# B&R Automation Studio project NewPendant_NG4_11_05_25A (part 4)

```c
	node[i].pHeadNode	= (UDINT)&node[P_MODE_TVL_CALIB];
	node[i].Type = N_EDIT;
	node[i].var.Type = T_SCALED;
	node[i].var.Var1ID = parGEN_CalibTime4;
	//strcpy(node[i++].var.Format, "(4)Time High Vel. REV:   %s");
	strcpy(node[i++].var.Format, "%name%: %s");

	node[i].pHeadNode	= (UDINT)&node[P_MODE_TVL_CALIB];
	node[i].Type = N_SCROLL +  N_EVENT ;
	node[i].Event = EVNT_OK;
	node[i].var.Type = T_STRING;
	node[i].var.Var1ID = (h++);
	strcpy(node[i++].var.Format, " %s");

	// P_MODE_TVL_CALIB_VER
	i= P_MODE_TVL_CALIB_VER;			h=varSTRING_HMI_0;
	SetPageDict(&cfg->PagesDict[n++] , P_MODE_TVL_CALIB_VER , "P_MODE_TVL_CALIB_VER");

	node[i].pHeadNode	= (UDINT)&node[P_MODE_TVL_CALIB_VER];
	node[i].Type = N_SCROLL +  N_EVENT ;
	node[i].Event = EVNT_CANCEL;
	strcpy(node[i++].var.Format, "Repeat !!!");	//ActPos:

	node[i].pHeadNode	= (UDINT)&node[P_MODE_TVL_CALIB_VER];
	node[i].Type = N_SCROLL;
	node[i].var.Type = T_STRING;
	node[i].var.Var1ID = (h++);
	strcpy(node[i++].var.Format, "%s");

	node[i].pHeadNode	= (UDINT)&node[P_MODE_TVL_CALIB_VER];
	node[i].Type = N_SCROLL;
	node[i].var.Type = T_STRING;
	node[i].var.Var1ID = (h++);
	strcpy(node[i++].var.Format, "%s");

	node[i].pHeadNode	= (UDINT)&node[P_MODE_TVL_CALIB_VER];
	node[i].Type = N_SCROLL;
	node[i].var.Type = T_STRING;
	node[i].var.Var1ID = (h++);
	strcpy(node[i++].var.Format, "%s");

	node[i].pHeadNode	= (UDINT)&node[P_MODE_TVL_CALIB_VER];
	node[i].Type = N_SCROLL +  N_EVENT ;
	node[i].Event = EVNT_OK;
	//node[i].var.Type = T_STRING;
	//node[i].var.Var1ID = (h++);
	//strcpy(node[i++].var.Format, "%s");
	strcpy(node[i++].var.Format, "Save Calibration !!!");

	///////////////////////////////////////

	i= P_MODE_TRACK_CALIB_PAR;			h=varSTRING_HMI_0;
	SetPageDict(&cfg->PagesDict[n++] , P_MODE_TRACK_CALIB_PAR , "P_MODE_TRACK_CALIB_PAR");

	node[i].pHeadNode	= (UDINT)&node[P_MODE_TRACK_CALIB_PAR];
	node[i].Type = N_SCROLL + N_EVENT;
	node[i].Event = EVNT_CANCEL;
	node[i].var.Type = T_STRING;
	node[i].var.Var1ID = (h++);
	strcpy(node[i++].var.Format, "%s");

	node[i].pHeadNode	= (UDINT)&node[P_MODE_TRACK_CALIB_PAR];
	node[i].Type = N_SCROLL + N_EDIT_IN_PLACE;
	node[i].var.Type = T_STRING;
	node[i].var.Var1ID = (h++);
	strcpy(node[i++].var.Format, "%s");

	node[i].pHeadNode	= (UDINT)&node[P_MODE_TRACK_CALIB_PAR];
	node[i].Type = N_EDIT;
	node[i].var.Type = T_SCALED;
	node[i].var.Var1ID = parGEN_Radius;
	strcpy(node[i++].var.Format, "%name%: %s");

	node[i].pHeadNode	= (UDINT)&node[P_MODE_TRACK_CALIB_PAR];
	node[i].Type = N_EDIT;
	node[i].var.Type = T_SCALED;
	node[i].var.Var1ID = parTVL_POS_OFFSET;
	strcpy(node[i++].var.Format, "%name%: %s");

	node[i].pHeadNode	= (UDINT)&node[P_MODE_TRACK_CALIB_PAR];
	node[i].Type = N_SCROLL + N_EVENT;
	node[i].Event = EVNT_OK;
	node[i].var.Type = T_STRING;
	node[i].var.Var1ID = (h++);
	strcpy(node[i++].var.Format, "%s");

	node[i].pHeadNode	= (UDINT)&node[P_MODE_TRACK_CALIB_PAR];
	node[i].Type = N_SCROLL + N_EVENT;
	node[i].Event = EVNT_ACKN;
	node[i].var.Type = T_STRING;
	node[i].var.Var1ID = (h++);
	strcpy(node[i++].var.Format, "%s");

	// P_MODE_TRACK_CALIB_PAR
	i= P_MODE_TRACK_CALIB;			h=varSTRING_HMI_0;
	SetPageDict(&cfg->PagesDict[n++] , P_MODE_TRACK_CALIB, "P_MODE_TRACK_CALIB");

	node[i].pHeadNode	= (UDINT)&node[P_MODE_TRACK_CALIB];
	node[i].Type = N_SCROLL + N_EVENT;
	node[i].Event = EVNT_CANCEL;
	node[i].var.Type = T_STRING;
	node[i].var.Var1ID = (h++);
	strcpy(node[i++].var.Format, "%s");

	node[i].pHeadNode	= (UDINT)&node[P_MODE_TRACK_CALIB];
	node[i].Type = N_SCROLL + N_EVENT;
	node[i].Event = EVNT_ACKN;
	node[i].var.Type = T_STRING;
	node[i].var.Var1ID = (h++);
	strcpy(node[i++].var.Format, "%s");

	node[i].pHeadNode	= (UDINT)&node[P_MODE_TRACK_CALIB];
	node[i].Type = N_SCROLL;
	node[i].var.Type = T_STRING;
	node[i].var.Var1ID = (h++);
	strcpy(node[i++].var.Format, "%s");

	node[i].pHeadNode	= (UDINT)&node[P_MODE_TRACK_CALIB];
	node[i].Type = N_SCROLL;
	node[i].var.Type = T_STRING;
	node[i].var.Var1ID = (h++);
	strcpy(node[i++].var.Format, "%s");

	node[i].pHeadNode	= (UDINT)&node[P_MODE_TRACK_CALIB];
	node[i].Type = N_SCROLL;
	node[i].var.Type = T_STRING;
	node[i].var.Var1ID = (h++);
	strcpy(node[i++].var.Format, "%s");

	node[i].pHeadNode	= (UDINT)&node[P_MODE_TRACK_CALIB];
	node[i].Type = N_SCROLL + N_EVENT;
	node[i].Event = EVNT_ACKN_ALL;
	node[i].var.Type = T_STRING;
	node[i].var.Var1ID = (h++);
	strcpy(node[i++].var.Format, "%s");

	node[i].pHeadNode	= (UDINT)&node[P_MODE_TRACK_CALIB];
	node[i].Type = N_SCROLL + N_EVENT;
	node[i].Event = EVNT_OK;
	node[i].var.Type = T_STRING;
	node[i].var.Var1ID = (h++);
	strcpy(node[i++].var.Format, "%s");

	// P_MODE_TRACK_CALIB_VER
	i= P_MODE_TRACK_CALIB_VER;			h=varSTRING_HMI_0;
	SetPageDict(&cfg->PagesDict[n++] , P_MODE_TRACK_CALIB_VER , "P_MODE_TRACK_CALIB_VER");

	node[i].pHeadNode	= (UDINT)&node[P_MODE_TRACK_CALIB_VER];
	node[i].Type = N_SCROLL + N_EVENT;
	node[i].Event = EVNT_CANCEL;
	node[i].var.Type = T_STRING;
	node[i].var.Var1ID = (h++);
	strcpy(node[i++].var.Format, "%s");

	node[i].pHeadNode	= (UDINT)&node[P_MODE_TRACK_CALIB_VER];
	node[i].Type = N_SCROLL + N_EVENT;
	node[i].Event = EVNT_ACKN;
	node[i].var.Type = T_STRING;
	node[i].var.Var1ID = (h++);
	strcpy(node[i++].var.Format, "%s");

	node[i].pHeadNode	= (UDINT)&node[P_MODE_TRACK_CALIB_VER];
	node[i].Type = N_SCROLL;
	node[i].var.Type = T_STRING;
	node[i].var.Var1ID = (h++);
	strcpy(node[i++].var.Format, "%s");

	node[i].pHeadNode	= (UDINT)&node[P_MODE_TRACK_CALIB_VER];
	node[i].Type = N_SCROLL;
	node[i].var.Type = T_STRING;
	node[i].var.Var1ID = (h++);
	strcpy(node[i++].var.Format, "%s");

	node[i].pHeadNode	= (UDINT)&node[P_MODE_TRACK_CALIB_VER];
	node[i].Type = N_SCROLL;
	node[i].var.Type = T_STRING;
	node[i].var.Var1ID = (h++);
	strcpy(node[i++].var.Format, "%s");

	node[i].pHeadNode	= (UDINT)&node[P_MODE_TRACK_CALIB_VER];
	node[i].Type = N_SCROLL + N_EVENT;
	node[i].Event = EVNT_OK;
	node[i].var.Type = T_STRING;
	node[i].var.Var1ID = (h++);
	strcpy(node[i++].var.Format, "%s");

	/////////////////////////////////////

	// P_SPEC_OPERATION
	i = P_SPEC_OPERATION;			h=varSTRING_HMI_0;
	SetPageDict(&cfg->PagesDict[n++] , P_SPEC_OPERATION , "P_SPEC_OPERATION");

	node[i].pHeadNode	= (UDINT)&node[P_SPEC_OPERATION];
	node[i].Type = N_JUMP;
	node[i].JumpLineID = 0;
	node[i].pJumpNode = (UDINT)&node[P_MENU];
	strcpy(node[i++].var.Format, " Return !!!");

	node[i].pHeadNode	= (UDINT)&node[P_SPEC_OPERATION];
	node[i].Type = N_SCROLL + N_EVENT;
	node[i].Event = EVNT_SET_AMERICAN_UNIT;
	strcpy(node[i++].var.Format, "Set Default Units !");

	node[i].pHeadNode	= (UDINT)&node[P_SPEC_OPERATION];
	node[i].Type = N_SCROLL + N_EVENT;
	node[i].Event = EVNT_SET_NORMAL_UNIT;
	strcpy(node[i++].var.Format, "Set SI Units !!!");

	node[i].pHeadNode	= (UDINT)&node[P_SPEC_OPERATION];
	node[i].Type = N_SCROLL + N_EVENT;
	node[i].Event = EVNT_LOAD_DEFAULT;
	strcpy(node[i++].var.Format, "Load Defaults !!!");

	node[i].pHeadNode	= (UDINT)&node[P_SPEC_OPERATION];
	node[i].Type = N_SCROLL + N_EVENT;
	node[i].Event = EVNT_LOAD_DEFAULT_CALIB;
	strcpy(node[i++].var.Format, "Load Default Calib !");

	node[i].pHeadNode	= (UDINT)&node[P_SPEC_OPERATION];
	node[i].Type = N_SCROLL + N_EVENT;
	node[i].Event = EVNT_ENT_BTN_REQ;
	strcpy(node[i++].var.Format, "Enter Btn Req!!");

	/** P_DIAGNOSTIC **/
	 i = P_DIAGNOSTIC;			h=varSTRING_HMI_0;
	SetPageDict(&cfg->PagesDict[n++] , P_DIAGNOSTIC , "P_DIAGNOSTIC");

	node[i].pHeadNode	= (UDINT)&node[P_DIAGNOSTIC];
	node[i].Type = N_SCROLL;
	node[i].var.Type = T_STRING;
	node[i].var.Var1ID = varSTRING_MasteStepTXT;
	strcpy(node[i++].var.Format, "M: %s");

	node[i].pHeadNode	= (UDINT)&node[P_DIAGNOSTIC];
	node[i].Type = N_JUMP;
	node[i].JumpLineID = 0;
	node[i].pJumpNode = (UDINT)&node[P_DIAGN_PROC];
	strcpy(node[i++].var.Format, "Diagn PROCESS");

	node[i].pHeadNode	= (UDINT)&node[P_DIAGNOSTIC];
	node[i].Type = N_JUMP;
	node[i].JumpLineID = 0;
	node[i].pJumpNode = (UDINT)&node[P_DIAGN_TML];
	strcpy(node[i++].var.Format, "Diagn TML Servo");

	node[i].pHeadNode	= (UDINT)&node[P_DIAGNOSTIC];
	node[i].Type = N_JUMP;
	node[i].JumpLineID = 0;
	node[i].pJumpNode = (UDINT)&node[P_DIAGN_DC_MTR];
	strcpy(node[i++].var.Format, "Diagn DC Mtrs");

	node[i].pHeadNode	= (UDINT)&node[P_DIAGNOSTIC];
	node[i].Type = N_JUMP;
	node[i].JumpLineID = 0;
	node[i].pJumpNode = (UDINT)&node[P_DIAGN_AXIS];
	strcpy(node[i++].var.Format, "Diagn Axises ");

	node[i].pHeadNode	= (UDINT)&node[P_DIAGNOSTIC];
	node[i].Type = N_JUMP;
	node[i].JumpLineID = 0;
	node[i].pJumpNode = (UDINT)&node[P_DIAGN_IO];
	strcpy(node[i++].var.Format, "Diagn I/O");

	node[i].pHeadNode	= (UDINT)&node[P_DIAGNOSTIC];
	node[i].Type = N_SCROLL + N_EVENT;
	node[i].Event = EVNT_RESTART ;
	node[i].var.Type = T_STRING;
	node[i].var.Var1ID = (h++);

	strcpy(node[i++].var.Format, "RESTART !!!");

	/** P_DIAGN_TML **/
	i = P_DIAGN_TML;			h=varSTRING_HMI_0;
	SetPageDict(&cfg->PagesDict[n++] , P_DIAGN_TML , "P_DIAGN_TML");

	node[i].pHeadNode	= (UDINT)&node[P_DIAGN_TML];
	node[i].Type = N_JUMP;
	node[i].JumpLineID = 0;
	node[i].pJumpNode = (UDINT)&node[P_DIAGNOSTIC];
	strcpy(node[i++].var.Format, " Return !!!");

	node[i].pHeadNode	= (UDINT)&node[P_DIAGN_TML];
	node[i].Type =    N_SCROLL + N_EDIT_IN_PLACE;
	node[i].var.Type = T_STRING;
	node[i].var.Var1ID = (h++);

	strcpy(node[i++].var.Format,"%s");

	node[i].pHeadNode	= (UDINT)&node[P_DIAGN_TML];
	node[i].Type = N_SCROLL + N_EDIT_IN_PLACE;
	node[i].var.Type = T_STRING;
	node[i].var.Var1ID = (h++);
	strcpy(node[i++].var.Format, "Stat: %s ");

	node[i].pHeadNode	= (UDINT)&node[P_DIAGN_TML];
	node[i].Type = N_SCROLL + N_EDIT_IN_PLACE;
	node[i].var.Var1ID = (h++);
	node[i].var.Type = T_STRING;
	strcpy(node[i++].var.Format, "%s");

	node[i].pHeadNode	= (UDINT)&node[P_DIAGN_TML];
	node[i].Type = N_SCROLL +	N_EVENT ;
	node[i].Event = EVNT_TOGGLE;
	node[i].var.Type = T_STRING;
	node[i].var.Var1ID = (h++);
	strcpy(node[i++].var.Format, "%s ");

	node[i].pHeadNode	= (UDINT)&node[P_DIAGN_TML];
	node[i].Type = N_SCROLL + N_EDIT_IN_PLACE;
	node[i].var.Type = T_STRING;
	node[i].var.Var1ID = (h++);
	strcpy(node[i++].var.Format, "%s");

	node[i].pHeadNode	= (UDINT)&node[P_DIAGN_TML];
	node[i].Type = N_SCROLL + N_EDIT_IN_PLACE;
	node[i].var.Type = T_STRING;
	node[i].var.Var1ID = (h++);
	strcpy(node[i++].var.Format, "%s");

	node[i].pHeadNode	= (UDINT)&node[P_DIAGN_TML];
	node[i].Type = N_SCROLL;
	node[i].var.Var1ID = (h++);
	node[i].var.Type = T_STRING;
	strcpy(node[i++].var.Format, "%s");

	node[i].pHeadNode	= (UDINT)&node[P_DIAGN_TML];
	node[i].Type = N_SCROLL;
	node[i].var.Type = T_STRING;
	node[i].var.Var1ID = (h++);
	strcpy(node[i++].var.Format, "EnInp: %s");

	node[i].pHeadNode	= (UDINT)&node[P_DIAGN_TML];
	node[i].Type = N_SCROLL;
	node[i].var.Type = T_STRING;
	node[i].var.Var1ID = (h++);
	strcpy(node[i++].var.Format, "%s "); // Inp 0 & 1

	node[i].pHeadNode	= (UDINT)&node[P_DIAGN_TML];
	node[i].Type = N_SCROLL;
	node[i].var.Type = T_STRING;
	node[i].var.Var1ID = (h++);
	strcpy(node[i++].var.Format, "%s "); //Inp 2 & 3

	node[i].pHeadNode	= (UDINT)&node[P_DIAGN_TML];
	node[i].Type = N_SCROLL;
	node[i].var.Type = T_STRING;
	node[i].var.Var1ID = (h++);
	strcpy(node[i++].var.Format, "%s "); //Out 0 & 1

	node[i].pHeadNode	= (UDINT)&node[P_DIAGN_TML];
	node[i].Type = N_SCROLL;
	node[i].var.Type = T_STRING;
	node[i].var.Var1ID = (h++);
	strcpy(node[i++].var.Format, "%s "); //Out 4

	node[i].pHeadNode	= (UDINT)&node[P_DIAGN_TML];
	node[i].Type = N_SCROLL;
	node[i].var.Type = T_STRING;
	node[i].var.Var1ID = (h++);
	strcpy(node[i++].var.Format, "xCMD: %s ");

	node[i].pHeadNode	= (UDINT)&node[P_DIAGN_TML];
	node[i].Type = N_SCROLL;
	node[i].var.Type = T_STRING;
	node[i].var.Var1ID = (h++);
	strcpy(node[i++].var.Format, "%s "); //Fbk:

	node[i].pHeadNode	= (UDINT)&node[P_DIAGN_TML];
	node[i].Type = N_SCROLL + N_EVENT;
	strcpy(node[i++].var.Format, "Jog Fwd");

	node[i].pHeadNode	= (UDINT)&node[P_DIAGN_TML];
	node[i].Type = N_SCROLL + N_EVENT;
	strcpy(node[i++].var.Format, "Jog Rev");

	node[i].pHeadNode	= (UDINT)&node[P_DIAGN_TML];
	node[i].Type = N_SCROLL + N_EVENT;
	node[i].Event = EVNT_OK;
	node[i].var.Type = T_STRING;
	node[i].var.Var1ID = (h++);
	strcpy(node[i++].var.Format, "Set ABS Home  !!!");

	node[i].pHeadNode	= (UDINT)&node[P_DIAGN_TML];
	node[i].Type = N_SCROLL + N_EVENT;
	node[i].Event = EVNT_LOAD;
	node[i].var.Type = T_STRING;
	node[i].var.Var1ID = (h++);
	strcpy(node[i++].var.Format, "LOAD Setup !!!");

	node[i].pHeadNode	= (UDINT)&node[P_DIAGN_TML];
	node[i].Type = N_SCROLL + N_EVENT;
	node[i].Event = EVNT_RESTART;
	node[i].var.Type = T_STRING;
	node[i].var.Var1ID = (h++);
	strcpy(node[i++].var.Format, "RESTART !!!");

	/** P_DIAGN_PROC **/
	i = P_DIAGN_PROC;			h=varSTRING_HMI_0;
	SetPageDict(&cfg->PagesDict[n++] , P_DIAGN_PROC , "P_DIAGN_PROC");

	node[i].pHeadNode	= (UDINT)&node[P_DIAGN_PROC];
	node[i].Type = N_JUMP;
	node[i].JumpLineID = 0;
	node[i].pJumpNode = (UDINT)&node[P_DIAGNOSTIC];
	strcpy(node[i++].var.Format, " Return !!!");

	node[i].pHeadNode	= (UDINT)&node[P_DIAGN_PROC];
	node[i].Type =    N_SCROLL + N_EDIT_IN_PLACE;
	node[i].var.Type = T_STRING;
	node[i].var.Var1ID = (h++);

	strcpy(node[i++].var.Format,"%s");

	node[i].pHeadNode	= (UDINT)&node[P_DIAGN_PROC];
	node[i].Type = N_SCROLL;
	node[i].var.Type = T_STRING;
	node[i].var.Var1ID = (h++);
	strcpy(node[i++].var.Format, "Stat: %s ");

	node[i].pHeadNode	= (UDINT)&node[P_DIAGN_PROC];
	node[i].Type = N_SCROLL;
	node[i].var.Type = T_STRING;
	node[i].var.Var1ID = (h++);
	strcpy(node[i++].var.Format, "%s ");

	node[i].pHeadNode	= (UDINT)&node[P_DIAGN_PROC];
	node[i].Type = N_SCROLL +	N_EVENT ;
	node[i].Event = EVNT_TOGGLE;
	node[i].var.Type = T_STRING;
	node[i].var.Var1ID = (h++);
	strcpy(node[i++].var.Format, "%s ");

	node[i].pHeadNode	= (UDINT)&node[P_DIAGN_PROC];
	node[i].Type = N_SCROLL + N_EVENT;
	node[i].Event = EVNT_RESTART ;
	node[i].var.Type = T_STRING;
	strcpy(node[i++].var.Format, "RESTART !!!");

	/** P_DIAGN_DC_MTR **/
	i = P_DIAGN_DC_MTR;			h=varSTRING_HMI_0;
	SetPageDict(&cfg->PagesDict[n++] , P_DIAGN_DC_MTR , "P_DIAGN_DC_MTR");

	node[i].pHeadNode	= (UDINT)&node[P_DIAGN_DC_MTR];
	node[i].Type = N_JUMP;
	node[i].JumpLineID = 0;
	node[i].pJumpNode = (UDINT)&node[P_DIAGNOSTIC];
	strcpy(node[i++].var.Format, " Return !!!");

	node[i].pHeadNode	= (UDINT)&node[P_DIAGN_DC_MTR];
	node[i].Type =    N_SCROLL + N_EDIT_IN_PLACE;
	node[i].var.Type = T_STRING;
	node[i].var.Var1ID = (h++);

	strcpy(node[i++].var.Format,"%s");

	node[i].pHeadNode	= (UDINT)&node[P_DIAGN_DC_MTR];
	node[i].Type = N_SCROLL;
	node[i].var.Type = T_STRING;
	node[i].var.Var1ID = (h++);
	strcpy(node[i++].var.Format, "%s ");

	node[i].pHeadNode	= (UDINT)&node[P_DIAGN_DC_MTR];
	node[i].Type = N_SCROLL +	N_EVENT ;
	node[i].Event = EVNT_TOGGLE;
	node[i].var.Type = T_STRING;
	node[i].var.Var1ID = (h++);
	strcpy(node[i++].var.Format, "%s ");

	node[i].pHeadNode	= (UDINT)&node[P_DIAGN_DC_MTR];
	node[i].Type = N_SCROLL;
	node[i].var.Type = T_STRING;
	node[i].var.Var1ID = (h++);
	strcpy(node[i++].var.Format, "Fbk: %s ");

	node[i].pHeadNode	= (UDINT)&node[P_DIAGN_DC_MTR];
	node[i].Type = N_SCROLL + N_EVENT;
	strcpy(node[i++].var.Format, "Jog Fwd");

	node[i].pHeadNode	= (UDINT)&node[P_DIAGN_DC_MTR];
	node[i].Type = N_SCROLL + N_EVENT;
	strcpy(node[i++].var.Format, "Jog Rev");

	/** P_DIAGN_AXIS **/
	i = P_DIAGN_AXIS;			h=varSTRING_HMI_0;
	SetPageDict(&cfg->PagesDict[n++] , P_DIAGN_AXIS , "P_DIAGN_AXIS");

	node[i].pHeadNode	= (UDINT)&node[P_DIAGN_AXIS];
	node[i].Type = N_JUMP;
	node[i].JumpLineID = 0;
	node[i].pJumpNode = (UDINT)&node[P_DIAGNOSTIC];
	strcpy(node[i++].var.Format, " Return !!!");

	node[i].pHeadNode	= (UDINT)&node[P_DIAGN_AXIS];
	node[i].Type =    N_SCROLL + N_EDIT_IN_PLACE;
	node[i].var.Type = T_STRING;
	node[i].var.Var1ID = (h++);

	strcpy(node[i++].var.Format,"%s");

	node[i].pHeadNode	= (UDINT)&node[P_DIAGN_AXIS];
	node[i].Type = N_SCROLL;
	node[i].var.Type = T_STRING;
	node[i].var.Var1ID = (h++);
	strcpy(node[i++].var.Format, "%s ");

	node[i].pHeadNode	= (UDINT)&node[P_DIAGN_AXIS];
	node[i].Type = N_SCROLL ;
	node[i].var.Type = T_STRING;
	node[i].var.Var1ID = (h++);
	strcpy(node[i++].var.Format, "%s ");

	node[i].pHeadNode	= (UDINT)&node[P_DIAGN_AXIS];
	node[i].Type = N_SCROLL ;
	node[i].var.Type = T_STRING;
	node[i].var.Var1ID = (h++);
	strcpy(node[i++].var.Format, "%s ");

	node[i].pHeadNode	= (UDINT)&node[P_DIAGN_AXIS];
	node[i].Type = N_SCROLL ;
	node[i].var.Type = T_STRING;
	node[i].var.Var1ID = (h++);
	strcpy(node[i++].var.Format, "%s ");

	/** P_DIAGN_IO **/
	i = P_DIAGN_IO;			h=varSTRING_HMI_0;
	SetPageDict(&cfg->PagesDict[n++] , P_DIAGN_IO , "P_DIAGN_IO");

	node[i].pHeadNode	= (UDINT)&node[P_DIAGN_IO];
	node[i].Type = N_JUMP;
	node[i].JumpLineID = 0;
	node[i].pJumpNode = (UDINT)&node[P_DIAGNOSTIC];
	strcpy(node[i++].var.Format, " Return !!!");

	node[i].pHeadNode	= (UDINT)&node[P_DIAGN_IO];
	node[i].Type = N_SCROLL;
	node[i].var.Var1ID = (h++);
	node[i].var.Type = T_STRING;

	strcpy(node[i++].var.Format, "%s");

	node[i].pHeadNode	= (UDINT)&node[P_DIAGN_IO];
	node[i].Type = N_SCROLL;
	node[i].var.Var1ID = (h++);
	node[i].var.Type = T_STRING;
	strcpy(node[i++].var.Format, "%s");

	node[i].pHeadNode	= (UDINT)&node[P_DIAGN_IO];
	node[i].Type = N_SCROLL;
	node[i].var.Var1ID = (h++);
	node[i].var.Type = T_STRING;
	strcpy(node[i++].var.Format, "%s");

	node[i].pHeadNode	= (UDINT)&node[P_DIAGN_IO];
	node[i].Type = N_SCROLL;
	node[i].var.Var1ID = (h++);
	node[i].var.Type = T_STRING;
	strcpy(node[i++].var.Format, "%s");

	node[i].pHeadNode	= (UDINT)&node[P_DIAGN_IO];
	node[i].Type = N_SCROLL;
	node[i].var.Var1ID = (h++);
	node[i].var.Type = T_STRING;
	strcpy(node[i++].var.Format, "%s");

	node[i].pHeadNode	= (UDINT)&node[P_DIAGN_IO];
	node[i].Type = N_SCROLL;
	node[i].var.Var1ID = (h++);
	node[i].var.Type = T_STRING;
	strcpy(node[i++].var.Format, "%s");

	node[i].pHeadNode	= (UDINT)&node[P_DIAGN_IO];
	node[i].Type = N_SCROLL;
	node[i].var.Var1ID = (h++);
	node[i].var.Type = T_STRING;
	strcpy(node[i++].var.Format, "%s");

	node[i].pHeadNode	= (UDINT)&node[P_DIAGN_IO];
	node[i].Type = N_SCROLL;
	node[i].var.Var1ID = (h++);
	node[i].var.Type = T_STRING;
	strcpy(node[i++].var.Format, "%s");

	node[i].pHeadNode	= (UDINT)&node[P_DIAGN_IO];
	node[i].Type = N_SCROLL;
	node[i].var.Var1ID = (h++);
	node[i].var.Type = T_STRING;
	strcpy(node[i++].var.Format, "%s");

	node[i].pHeadNode	= (UDINT)&node[P_DIAGN_IO];
	node[i].Type = N_SCROLL;
	node[i].var.Var1ID = (h++);
	node[i].var.Type = T_STRING;
	strcpy(node[i++].var.Format, "%s");

	node[i].pHeadNode	= (UDINT)&node[P_DIAGN_IO];
	node[i].Type = N_SCROLL;
	node[i].var.Var1ID = (h++);
	node[i].var.Type = T_STRING;
	strcpy(node[i++].var.Format, "%s");

	/** P_LOGS **/
	 i = P_LOGS;			h=varSTRING_HMI_0;
	SetPageDict(&cfg->PagesDict[n++] , P_LOGS , "P_LOGS");

	node[i].pHeadNode	= (UDINT)&node[P_LOGS];
	node[i].Type = N_SCROLL + N_EDIT_IN_PLACE;
	node[i].var.Var1ID = (h++);
	node[i].var.Type = T_STRING;
	strcpy(node[i++].var.Format, "%s");

	node[i].pHeadNode	= (UDINT)&node[P_LOGS];
	node[i].Type = N_SCROLL + N_EDIT_IN_PLACE;
	node[i].var.Var1ID = (h++);
	node[i].var.Type = T_STRING;
	strcpy(node[i++].var.Format, "%s");

	node[i].pHeadNode	= (UDINT)&node[P_LOGS];
	node[i].Type = N_SCROLL + N_EDIT_IN_PLACE;
	node[i].var.Var1ID = (h++);
	node[i].var.Type = T_STRING;
	strcpy(node[i++].var.Format, "%s");

	node[i].pHeadNode	= (UDINT)&node[P_LOGS];
	node[i].Type = N_SCROLL + N_EDIT_IN_PLACE;
	node[i].var.Var1ID = (h++);
	node[i].var.Type = T_STRING;
	strcpy(node[i++].var.Format, "%s");

	node[i].pHeadNode	= (UDINT)&node[P_LOGS];
	node[i].Type = N_SCROLL + N_EDIT_IN_PLACE;
	node[i].var.Var1ID = (h++);
	node[i].var.Type = T_STRING;
	strcpy(node[i++].var.Format, "%s");

	node[i].pHeadNode	= (UDINT)&node[P_LOGS];
	node[i].Type = N_SCROLL + N_EDIT_IN_PLACE;
	node[i].var.Var1ID = (h++);
	node[i].var.Type = T_STRING;
	strcpy(node[i++].var.Format, "%s");

	/** P_ERRORS **/
	 i = P_ERRORS;			h=varSTRING_HMI_0;
	SetPageDict(&cfg->PagesDict[n++] , P_ERRORS , "P_ERRORS");

	node[i].pHeadNode	= (UDINT)&node[P_ERRORS];
	node[i].Type = N_SCROLL + N_EDIT_IN_PLACE;
	node[i].var.Var1ID = (h++);
	node[i].var.Type = T_STRING;
	strcpy(node[i++].var.Format, "%s");

	node[i].pHeadNode	= (UDINT)&node[P_ERRORS];
	node[i].Type = N_SCROLL + N_EDIT_IN_PLACE;
	node[i].var.Var1ID = (h++);
	node[i].var.Type = T_STRING;
	strcpy(node[i++].var.Format, "%s");

	node[i].pHeadNode	= (UDINT)&node[P_ERRORS];
	node[i].Type = N_SCROLL + N_EDIT_IN_PLACE;
	node[i].var.Var1ID = (h++);
	node[i].var.Type = T_STRING;
	strcpy(node[i++].var.Format, "  %s");

	node[i].pHeadNode	= (UDINT)&node[P_ERRORS];
	node[i].Type = N_SCROLL + N_EDIT_IN_PLACE;
	node[i].var.Var1ID = (h++);
	node[i].var.Type = T_STRING;
	strcpy(node[i++].var.Format, "  %s");

	node[i].pHeadNode	= (UDINT)&node[P_ERRORS];
	node[i].Type = N_SCROLL + N_EDIT_IN_PLACE;
	node[i].var.Var1ID = (h++);
	node[i].var.Type = T_STRING;
	strcpy(node[i++].var.Format, "  %s");

	node[i].pHeadNode	= (UDINT)&node[P_ERRORS];
	node[i].Type = N_SCROLL + N_EVENT;
	node[i].Event = EVNT_ACKN_ALL;
	strcpy(node[i++].var.Format, " ACK All Errors !!!");

	//////////////////////////////////////////////////////////
	//////////    FOR TESTING ONLY -

	/** P_PAR_REVIEW **/
	i = P_PAR_REVIEW;			h=varSTRING_HMI_0;
	SetPageDict(&cfg->PagesDict[n++] , P_PAR_REVIEW , "P_PAR_REVIEW");

	node[i].pHeadNode	= (UDINT)&node[P_PAR_REVIEW];
	node[i].Type = N_JUMP;
	node[i].JumpLineID = 0;
	node[i].pJumpNode = (UDINT)&node[P_MENU];
	strcpy(node[i++].var.Format, "Return ");

	node[i].pHeadNode	= (UDINT)&node[P_PAR_REVIEW];
	node[i].Type = N_SCROLL;
	strcpy(node[i++].var.Format, "**** AVC *****");

	node[i].pHeadNode	= (UDINT)&node[P_PAR_REVIEW];
	node[i].Type = N_EDIT;
	node[i].MinUserLevel = USER_OPERATOR;
	node[i].var.Type = T_SCALED;
	node[i].var.Var1ID = parAVC_StartDly;
	//strcpy(node[i++].var.Format, "AVC UpslopeDly %s");
	strcpy(node[i++].var.Format, "%name%: %s");

	node[i].pHeadNode	= (UDINT)&node[P_PAR_REVIEW];
	node[i].Type = N_EDIT;
	node[i].MinUserLevel = USER_OPERATOR;
	node[i].var.Type = T_SCALED;
	node[i].var.Var1ID = parAVC_Upslope;
	//strcpy(node[i++].var.Format, "AVC Upslope %s");
	strcpy(node[i++].var.Format, "%name%: %s");

	node[i].pHeadNode	= (UDINT)&node[P_PAR_REVIEW];
	node[i].Type = N_EDIT;
	node[i].MinUserLevel = USER_OPERATOR;
	node[i].var.Type = T_SCALED;
	node[i].var.Var1ID = parAVC_StopDly;
	//strcpy(node[i++].var.Format, "AVC StopDly %s");
	strcpy(node[i++].var.Format, "%name%: %s");

	node[i].pHeadNode	= (UDINT)&node[P_PAR_REVIEW];
	node[i].Type = N_EDIT;
	node[i].MinUserLevel = USER_OPERATOR;
	node[i].var.Type = T_SCALED;
	node[i].var.Var1ID = parAVC_DownSlope;
	//strcpy(node[i++].var.Format, "AVC DownSlope %s");
	strcpy(node[i++].var.Format, "%name%: %s");

	node[i].pHeadNode	= (UDINT)&node[P_PAR_REVIEW];
	node[i].Type = N_EDIT;
	node[i].MinUserLevel = USER_OPERATOR;
	node[i].var.Type = T_SCALED;
	node[i].var.Var1ID = parAVC_HoldTm;
	//strcpy(node[i++].var.Format, "AVC HoldTm %s");
	strcpy(node[i++].var.Format, "%name%: %s");

	node[i].pHeadNode	= (UDINT)&node[P_PAR_REVIEW];
	node[i].Type = N_SCROLL;
	strcpy(node[i++].var.Format, "**** TVL *****");

	node[i].pHeadNode	= (UDINT)&node[P_PAR_REVIEW];
	node[i].Type = N_EDIT;
	node[i].MinUserLevel = USER_OPERATOR;
	node[i].var.Type = T_SCALED;
	node[i].var.Var1ID = parTVL_StartDly;
	//strcpy(node[i++].var.Format, "TVL_StartDly %s");
	strcpy(node[i++].var.Format, "%name%: %s");

	node[i].pHeadNode	= (UDINT)&node[P_PAR_REVIEW];
	node[i].Type = N_EDIT;
	node[i].MinUserLevel = USER_OPERATOR;
	node[i].var.Type = T_SCALED;
	node[i].var.Var1ID = parTVL_RampUp;
	//strcpy(node[i++].var.Format, "TVL RampUp %s");
	strcpy(node[i++].var.Format, "%name%: %s");

	node[i].pHeadNode	= (UDINT)&node[P_PAR_REVIEW];
	node[i].Type = N_EDIT;
	node[i].MinUserLevel = USER_OPERATOR;
	node[i].var.Type = T_SCALED;
	node[i].var.Var1ID = parTVL_StopDly;
	//strcpy(node[i++].var.Format, "TVL StopDly %s");
	strcpy(node[i++].var.Format, "%name%: %s");

	node[i].pHeadNode	= (UDINT)&node[P_PAR_REVIEW];
	node[i].Type = N_EDIT;
	node[i].MinUserLevel = USER_OPERATOR;
	node[i].var.Type = T_SCALED;
	node[i].var.Var1ID = parTVL_RampDwn;
	//strcpy(node[i++].var.Format, "TVL RampDwn %s");
	strcpy(node[i++].var.Format, "%name%: %s");

	node[i].pHeadNode	= (UDINT)&node[P_PAR_REVIEW];
	node[i].Type = N_EDIT;
	node[i].MinUserLevel = USER_OPERATOR;
	node[i].var.Type = T_SCALED;
	node[i].var.Var1ID = parTVL_RewrapDly;
	//strcpy(node[i++].var.Format, "TVL RewrapDly %s");
	strcpy(node[i++].var.Format, "%name%: %s");

	node[i].pHeadNode	= (UDINT)&node[P_PAR_REVIEW];
	node[i].Type = N_EDIT;
	node[i].MinUserLevel = USER_OPERATOR;
	node[i].var.Type = T_SCALED;
	node[i].var.Var1ID = parTVL_OverlapDist;
	//strcpy(node[i++].var.Format, "TVL Overlap %s");
	strcpy(node[i++].var.Format, "%name%: %s");

	node[i].pHeadNode	= (UDINT)&node[P_PAR_REVIEW];
	node[i].Type = N_SCROLL;
	strcpy(node[i++].var.Format, "**** TIG AMP *****");

	node[i].pHeadNode	= (UDINT)&node[P_PAR_REVIEW];
	node[i].Type = N_EDIT;
	node[i].MinUserLevel = USER_OPERATOR;
	node[i].var.Type = T_SCALED;
	node[i].var.Var1ID = parTIG_StartDly;
	//strcpy(node[i++].var.Format, "TIG StartDly %s");
	strcpy(node[i++].var.Format, "%name%: %s");

	node[i].pHeadNode	= (UDINT)&node[P_PAR_REVIEW];
	node[i].Type = N_EDIT;
	node[i].MinUserLevel = USER_OPERATOR;
	node[i].var.Type = T_SCALED;
	node[i].var.Var1ID = parTIG_RampUp;
	//strcpy(node[i++].var.Format, "TIG RampUp %s");
	strcpy(node[i++].var.Format, "%name%: %s");

	node[i].pHeadNode	= (UDINT)&node[P_PAR_REVIEW];
	node[i].Type = N_EDIT;
	node[i].MinUserLevel = USER_OPERATOR;
	node[i].var.Type = T_SCALED;
	node[i].var.Var1ID = parTIG_StopDly;
	//strcpy(node[i++].var.Format, "TIG StopDly %s");
	strcpy(node[i++].var.Format, "%name%: %s");

	node[i].pHeadNode	= (UDINT)&node[P_PAR_REVIEW];
	node[i].Type = N_EDIT;
	node[i].MinUserLevel = USER_OPERATOR;
	node[i].var.Type = T_SCALED;
	node[i].var.Var1ID = parTIG_RampDwn;
	//strcpy(node[i++].var.Format, "TIG RampDwn %s");
	strcpy(node[i++].var.Format, "%name%: %s");

	node[i].pHeadNode	= (UDINT)&node[P_PAR_REVIEW];
	node[i].Type = N_SCROLL;
	strcpy(node[i++].var.Format, "**** OSC *****");

	node[i].pHeadNode	= (UDINT)&node[P_PAR_REVIEW];
	node[i].Type = N_EDIT;
	node[i].MinUserLevel = USER_OPERATOR;
	node[i].var.Type = T_SCALED;
	node[i].var.Var1ID = parOSC_StartDly;
	//strcpy(node[i++].var.Format, "OSC StartDly %s");
	strcpy(node[i++].var.Format, "%name%: %s");

	node[i].pHeadNode	= (UDINT)&node[P_PAR_REVIEW];
	node[i].Type = N_EDIT;
	node[i].MinUserLevel = USER_OPERATOR;
	node[i].var.Type = T_SCALED;
	node[i].var.Var1ID = parOSC_RampUp;
	//strcpy(node[i++].var.Format, "OSC RampUp %s");
	strcpy(node[i++].var.Format, "%name%: %s");

	node[i].pHeadNode	= (UDINT)&node[P_PAR_REVIEW];
	node[i].Type = N_EDIT;
	node[i].MinUserLevel = USER_OPERATOR;
	node[i].var.Type = T_SCALED;
	node[i].var.Var1ID = parOSC_StopDly;
	//strcpy(node[i++].var.Format, "OSC StopDly %s");
	strcpy(node[i++].var.Format, "%name%: %s");

	node[i].pHeadNode	= (UDINT)&node[P_PAR_REVIEW];
	node[i].Type = N_EDIT;
	node[i].MinUserLevel = USER_OPERATOR;
	node[i].var.Type = T_SCALED;
	node[i].var.Var1ID = parOSC_RampDwn;
	//strcpy(node[i++].var.Format, "OSC RampDwn %s");
	strcpy(node[i++].var.Format, "%name%: %s");

	node[i].pHeadNode	= (UDINT)&node[P_PAR_REVIEW];
	node[i].Type = N_SCROLL;
	strcpy(node[i++].var.Format, "**** WF *****");

	node[i].pHeadNode	= (UDINT)&node[P_PAR_REVIEW];
	node[i].Type = N_EDIT;
	node[i].MinUserLevel = USER_OPERATOR;
	node[i].var.Type = T_SCALED;
	node[i].var.Var1ID = parWF_StartDly;
	//strcpy(node[i++].var.Format, "parWF StartDly %s");
	strcpy(node[i++].var.Format, "%name%: %s");

	node[i].pHeadNode	= (UDINT)&node[P_PAR_REVIEW];
	node[i].Type = N_EDIT;
	node[i].MinUserLevel = USER_OPERATOR;
	node[i].var.Type = T_SCALED;
	node[i].var.Var1ID = parWF_RampUp;
	//strcpy(node[i++].var.Format, "WF RampUp %s");
	strcpy(node[i++].var.Format, "%name%: %s");

	node[i].pHeadNode	= (UDINT)&node[P_PAR_REVIEW];
	node[i].Type = N_EDIT;
	node[i].MinUserLevel = USER_OPERATOR;
	node[i].var.Type = T_SCALED;
	node[i].var.Var1ID = parWF_StopDly;
	//strcpy(node[i++].var.Format, "WF StopDly %s");
	strcpy(node[i++].var.Format, "%name%: %s");

	node[i].pHeadNode	= (UDINT)&node[P_PAR_REVIEW];
	node[i].Type = N_EDIT;
	node[i].MinUserLevel = USER_OPERATOR;
	node[i].var.Type = T_SCALED;
	node[i].var.Var1ID = parWF_RampDwn;
	//strcpy(node[i++].var.Format, "WF RampDwn %s");
	strcpy(node[i++].var.Format, "%name%: %s");

	node[i].pHeadNode	= (UDINT)&node[P_PAR_REVIEW];
	node[i].Type = N_SCROLL;
	strcpy(node[i++].var.Format, "**** WP *****");

	node[i].pHeadNode	= (UDINT)&node[P_PAR_REVIEW];
	node[i].Type = N_EDIT;
	node[i].MinUserLevel = USER_OPERATOR;
	node[i].var.Type = T_SCALED;
	node[i].var.Var1ID = parWP_StartDly;
	//strcpy(node[i++].var.Format, "WP StartDly %s");
	strcpy(node[i++].var.Format, "%name%: %s");

	node[i].pHeadNode	= (UDINT)&node[P_PAR_REVIEW];
	node[i].Type = N_EDIT;
	node[i].MinUserLevel = USER_OPERATOR;
	node[i].var.Type = T_SCALED;
	node[i].var.Var1ID = parWP_RampUp;
	//strcpy(node[i++].var.Format, "WP RampUp %s");
	strcpy(node[i++].var.Format, "%name%: %s");

	node[i].pHeadNode	= (UDINT)&node[P_PAR_REVIEW];
	node[i].Type = N_EDIT;
	node[i].MinUserLevel = USER_OPERATOR;
	node[i].var.Type = T_SCALED;
	node[i].var.Var1ID = parWP_StopDly;
	//strcpy(node[i++].var.Format, "WP StopDly %s");
	strcpy(node[i++].var.Format, "%name%: %s");

	node[i].pHeadNode	= (UDINT)&node[P_PAR_REVIEW];
	node[i].Type = N_EDIT;
	node[i].MinUserLevel = USER_OPERATOR;
	node[i].var.Type = T_SCALED;
	node[i].var.Var1ID = parWP_RampDwn;
	//strcpy(node[i++].var.Format, "WP RampDwn %s");
	strcpy(node[i++].var.Format, "%name%: %s");

	node[i].pHeadNode	= (UDINT)&node[P_PAR_REVIEW];
	node[i].Type = N_SCROLL;
	strcpy(node[i++].var.Format, "**** HW *****");

	node[i].pHeadNode	= (UDINT)&node[P_PAR_REVIEW];
	node[i].Type = N_EDIT;
	node[i].MinUserLevel = USER_OPERATOR;
	node[i].var.Type = T_SCALED;
	node[i].var.Var1ID = parHW_RampUpDly;
	//strcpy(node[i++].var.Format, "HW RampUpDly %s");
	strcpy(node[i++].var.Format, "%name%: %s");

	node[i].pHeadNode	= (UDINT)&node[P_PAR_REVIEW];
	node[i].Type = N_EDIT;
	node[i].MinUserLevel = USER_OPERATOR;
	node[i].var.Type = T_SCALED;
	node[i].var.Var1ID = parHW_RampUp;
	//strcpy(node[i++].var.Format, "HW RampUp %s");
	strcpy(node[i++].var.Format, "%name%: %s");

	node[i].pHeadNode	= (UDINT)&node[P_PAR_REVIEW];
	node[i].Type = N_EDIT;
	node[i].MinUserLevel = USER_OPERATOR;
	node[i].var.Type = T_SCALED;
	node[i].var.Var1ID = parHW_RampDwnDly;
	//strcpy(node[i++].var.Format, "HW RampDwnDly %s");
	strcpy(node[i++].var.Format, "%name%: %s");

	node[i].pHeadNode	= (UDINT)&node[P_PAR_REVIEW];
	node[i].Type = N_EDIT;
	node[i].MinUserLevel = USER_OPERATOR;
	node[i].var.Type = T_SCALED;
	node[i].var.Var1ID = parHW_RampDwn;
	//strcpy(node[i++].var.Format, "HW RampDwn %s");
	strcpy(node[i++].var.Format, "%name%: %s");

	node[i].pHeadNode	= (UDINT)&node[P_PAR_REVIEW];
	node[i].Type = N_SCROLL;
	strcpy(node[i++].var.Format, "**** GAS *****");

	node[i].pHeadNode	= (UDINT)&node[P_PAR_REVIEW];
	node[i].Type = N_EDIT;
	node[i].MinUserLevel = USER_OPERATOR;
	node[i].var.Type = T_SCALED;
	node[i].var.Var1ID = parGAS_PrePurgeTm;
	//strcpy(node[i++].var.Format, "GAS PrePurgeTm %s");
	strcpy(node[i++].var.Format, "%name%: %s");

	node[i].pHeadNode	= (UDINT)&node[P_PAR_REVIEW];
	node[i].Type = N_EDIT;
	node[i].MinUserLevel = USER_OPERATOR;
	node[i].var.Type = T_SCALED;
	node[i].var.Var1ID = parGAS_PostPurgeTm;
	//strcpy(node[i++].var.Format, "GAS PostPurgeTm %s");
	strcpy(node[i++].var.Format, "%name%: %s");

	//////////////////////////////////////////////////////////

	m->nodesNum[0] = nodeNum;

	/////////////////////////
	// Populate nodes ID //////
	for(i = 0 ; i < nodeNum ; i ++){
		node[i].ID = (UINT)i;

		// Sanitary - remove old absolete attributes - just in case
		node[i].Type = node[i].Type & (0xFFFF - (N_EDIT_DIS + N_NO_PREFIX + N_USER_EDIT + N_ONLY_LCD));

	}

	// Populate HeadID
	for(i = 0 ; i < nodeNum ; i ++){

		if(	node[i].pHeadNode){
			tempNode  = (LCD_NODE_obj*)node[i].pHeadNode;

			if(tempNode)
				node[i].HeadID = tempNode->ID;
		}
		else
			node[i].pHeadNode = 0;
	}

	// Populate JumpNodeID
	for(i = 0 ; i < nodeNum ; i ++){

		tempNode = (LCD_NODE_obj*)node[i].pJumpNode;

		if(tempNode)
			node[i].JumpNodeID = tempNode->ID;

	}

}

void HardCodeCFg(MASTER_typ *m){

int i, k;
char status;
Cfg_typ *cfg;
CurCfg_typ *curCfg;
Scaled_Var_obj *var;
CurCalib_typ *defCalib , *calib;

	if(!m)
		return;

	cfg = (Cfg_typ*) m->pCfg;
	curCfg = (CurCfg_typ*) m->pCurCfg;
	var = (Scaled_Var_obj*) m->pScaledVar;
	defCalib =  (CurCalib_typ*) m->pDefaultCalib;
	calib =	(CurCalib_typ*) m->pCalib;

	if(!cfg || ! curCfg || !var || !defCalib || !calib)
		return;

	//////////////////////////////////////////////////////
	//   Button Mode when edit value  - 1.- hold button
	i = parLCD_BtnMode;
	strcpy(var[i].name , "Edit Button Mode");
	strcpy(var[i].enumTXT, "parLCD_BtnMode");
	var[i].PlcUnitIndx = unitIU;
	var[i].unitType = unitIU;
	var[i].DefaultUnit = unitIU;
	var[i].precision = 2;
	cfg->Param[i].min = 0.0;
	cfg->Param[i].max = 1.0;
	cfg->Param[i].incrMin = 1.0;
	cfg->Param[i].incrMax = 1.0;
	cfg->Param[i].defaultVal = 1.0;
	var[i].segm = 0;

	//////////////////////////////////////////////////////
	//   OSCILLATION

	i = parOSC_Indx_Vel;
	strcpy(var[i].name , "OSC Index Speed");
	strcpy(var[i].enumTXT, "parOSC_Indx_Vel");
	var[i].PlcUnitIndx = unitIU;
	var[i].unitType = unitSpeed;
	var[i].DefaultUnit = UNIT_inch_per_sec;
	var[i].precision = 0;
	cfg->Param[i].min = 0.01 * in_2_mm / 1.0;
	cfg->Param[i].max = 1.0 * in_2_mm / 1.0;
	cfg->Param[i].incrMin = 0.01 * in_2_mm / 1.0;
	cfg->Param[i].incrMax = 5 * cfg->Param[i].incrMin;
	cfg->Param[i].defaultVal = 0.25 * in_2_mm / 1.0;
	var[i].segm = 0;

	i = parOSC_StartDly;
	strcpy(var[i].name , "OSC START DLY");
	strcpy(var[i].enumTXT, "parOSC_StartDly");
	var[i].PlcUnitIndx = unitIU;
	var[i].unitType = unitTime;
	var[i].DefaultUnit = UNIT_sec;
	var[i].precision = 1;
	cfg->Param[i].min = 0.0;
	cfg->Param[i].max = 60.0;
	cfg->Param[i].incrMin = 0.1;
	cfg->Param[i].incrMax = 1.0;
	cfg->Param[i].defaultVal = 2.0;
	var[i].segm = 0;

	i = parOSC_RampUp;
	strcpy(var[i].name , "OSC UPSLOPE TM");
	strcpy(var[i].enumTXT, "parOSC_RampUp");
	var[i].PlcUnitIndx = unitIU;
	var[i].unitType = unitTime;
	var[i].DefaultUnit = UNIT_sec;
	var[i].precision = 1;
	cfg->Param[i].min = 0.0;
	cfg->Param[i].max = 60.0;
	cfg->Param[i].incrMin = 0.1;
	cfg->Param[i].incrMax = 1.0;
	cfg->Param[i].defaultVal = 4.0;
	var[i].segm = 0;

	i = parOSC_Amplit;
	strcpy(var[i].name , "OSC WIDTH");
	strcpy(var[i].enumTXT, "parOSC_Amplit");
	var[i].PlcUnitIndx = unitIU;
	var[i].unitType = unitLength;
	var[i].DefaultUnit = UNIT_inch;
	var[i].precision = 1;
	cfg->Param[i].min = 0.0;
	// Was changed to 3 inch 12 June 2020 by Mark request
	cfg->Param[i].max = 3.0 * 25.4;
	cfg->Param[i].incrMin = 0.01 * in_2_mm;
	cfg->Param[i].incrMax = 1.0 * in_2_mm;
	cfg->Param[i].defaultVal = 0.35 * in_2_mm ;
	var[i].segm = 1;

	i = parOSC_FinalAmplit;
	strcpy(var[i].name , "OSC FINAL WIDTH");
	strcpy(var[i].enumTXT, "parOSC_FinalAmplit");
	var[i].PlcUnitIndx = unitIU;
	var[i].unitType = unitLength;
	var[i].DefaultUnit = UNIT_inch;
	var[i].precision = 1;
	cfg->Param[i].min = 0.0;
	cfg->Param[i].max = 25.4;
	cfg->Param[i].incrMin = 0.05 * in_2_mm;
	cfg->Param[i].incrMax = 1.0 * in_2_mm;
	cfg->Param[i].defaultVal = 0.05 * in_2_mm ; // 1/4 " = 6.35 mm
	var[i].segm = 0;

	i = parOSC_InitAmplit;
	strcpy(var[i].name , "OSC INITIAL WIDTH");
	strcpy(var[i].enumTXT, "parOSC_InitAmplit");
	var[i].PlcUnitIndx = unitIU;
	var[i].unitType = unitLength;
	var[i].DefaultUnit = UNIT_inch;
	var[i].precision = 1;
	cfg->Param[i].min = 0.0;
	cfg->Param[i].max = 25.4;
	cfg->Param[i].incrMin = 0.05 * in_2_mm;
	cfg->Param[i].incrMax = 1.0 * in_2_mm;
	cfg->Param[i].defaultVal = 0.0 * in_2_mm ; // 1/4 " = 6.35 mm
	var[i].segm = 0;

	i = parOSC_Indx;
	strcpy(var[i].name , "OSC Index");
	strcpy(var[i].enumTXT, "parOSC_Indx");
	var[i].PlcUnitIndx = unitIU;
	var[i].unitType = unitLength;
	var[i].DefaultUnit = UNIT_inch;
	var[i].precision = 1;
	cfg->Param[i].min = -25.4;
	cfg->Param[i].max = 25.4;
	cfg->Param[i].incrMin = 0.01 * in_2_mm;
	cfg->Param[i].incrMax = 1.0 * in_2_mm;
	cfg->Param[i].defaultVal = 0.25 * in_2_mm ; // 1/4 " = 6.35 mm
	var[i].segm = 0;

	i = parOSC_Period;
	strcpy(var[i].name , "OSC Period");
	strcpy(var[i].enumTXT, "parOSC_Period");
	var[i].PlcUnitIndx = unitIU;
	var[i].unitType =  unitIU;
	var[i].DefaultUnit = unitIU;
	var[i].precision = 0;
	cfg->Param[i].min = 0.0;
	cfg->Param[i].max = 100000.0;
	cfg->Param[i].incrMin = 1;
	cfg->Param[i].incrMax = 1;
	cfg->Param[i].defaultVal = 40;
	var[i].segm = 0;

	i = parOSC_StopDly;
	strcpy(var[i].name , "OSC DOWNSLOPE DLY");
	strcpy(var[i].enumTXT, "parOSC_StopDly");
	var[i].PlcUnitIndx = unitIU;
	var[i].unitType = unitTime;
	var[i].DefaultUnit = UNIT_sec;
	var[i].precision = 1;
	cfg->Param[i].min = 0.0;
	cfg->Param[i].max = 60.0;
	cfg->Param[i].incrMin = 0.1;
	cfg->Param[i].incrMax = 1.0;
	cfg->Param[i].defaultVal = 7.0;
	var[i].segm = 0;

	i = parOSC_RampDwn;
	strcpy(var[i].name , "OSC DOWNSLOPE TM");
	strcpy(var[i].enumTXT, "parOSC_RampDwn");
	var[i].PlcUnitIndx = unitIU;
	var[i].unitType = unitTime;
	var[i].DefaultUnit = UNIT_sec;
	var[i].precision = 1;
	cfg->Param[i].min = 0.0;
	cfg->Param[i].max = 60.0;
	cfg->Param[i].incrMin = 0.1;
	cfg->Param[i].incrMax = 1.0;
	cfg->Param[i].defaultVal = 1.0;
	var[i].segm = 0;

	i = parOSC_RampUpdate;
	strcpy(var[i].name , "Osc Ramp Update");
	strcpy(var[i].enumTXT, "parOSC_RampUpdate");
	var[i].PlcUnitIndx = unitIU;
	var[i].unitType = unitTime;
	var[i].DefaultUnit = UNIT_sec;
	var[i].precision = 1;
	cfg->Param[i].min = 0.0;
	cfg->Param[i].max = 60.0;
	cfg->Param[i].incrMin = 0.1;
	cfg->Param[i].incrMax = 1.0;
	cfg->Param[i].defaultVal = 0.1;
	var[i].segm = 0;

	i = parOSC_Excur;
	strcpy(var[i].name , "Osc Excursion");
	strcpy(var[i].enumTXT, "parOSC_Excur");
	var[i].PlcUnitIndx = unitIU;
	var[i].unitType = unitTime;
	var[i].DefaultUnit = UNIT_sec;
	var[i].precision = 1;
	cfg->Param[i].min = 0.05;
	cfg->Param[i].max = 10.0;
	cfg->Param[i].incrMin = 0.05;
	cfg->Param[i].incrMax = 1.0;
	cfg->Param[i].defaultVal = 1.0;
	var[i].segm = 1;

	i = parOSC_Dwell_In;
	strcpy(var[i].name , "Osc Dwell In");
	strcpy(var[i].enumTXT, "parOSC_Dwell_In");
	var[i].PlcUnitIndx = unitIU;
	var[i].unitType = unitTime;
	var[i].DefaultUnit = UNIT_sec;
	var[i].precision = 1;
	cfg->Param[i].min = 0.0;
	cfg->Param[i].max = 6.0;
	cfg->Param[i].incrMin = 0.1;
	cfg->Param[i].incrMax = 1.0;
	cfg->Param[i].defaultVal = 1.0;
	var[i].segm = 1;

	i = parOSC_Dwell_Out;
	strcpy(var[i].name , "Osc Dwell Out");
	strcpy(var[i].enumTXT, "parOSC_Dwell_Out");
	var[i].PlcUnitIndx = unitIU;
	var[i].unitType = unitTime;
	var[i].DefaultUnit = UNIT_sec;
	var[i].precision = 1;
	cfg->Param[i].min = 0.0;
	cfg->Param[i].max = 6.0;
	cfg->Param[i].incrMin = 0.1;
	cfg->Param[i].incrMax = 1.0;
	cfg->Param[i].defaultVal = 1.0;
	var[i].segm = 1;

	i = parOSC_JogSpeedDirCntrl;
	strcpy(var[i].name , "OSC Jog Speed");
	strcpy(var[i].enumTXT, "parOSC_JogSpeedDirCntrl");
	var[i].PlcUnitIndx = unitIU;
	var[i].unitType = unitPerc;
	var[i].DefaultUnit = UNIT_PERCENT;
	var[i].precision = 1;
	cfg->Param[i].min = 0.0;
	cfg->Param[i].max = 1.0;
	cfg->Param[i].incrMin = 0.05;
	cfg->Param[i].incrMax = 0.1;
	cfg->Param[i].defaultVal = 0.75;
	var[i].segm = 0;

	i = parOSC_JogSpeed;
	strcpy(var[i].name , "OSC Jog Speed");
	strcpy(var[i].enumTXT, "parOSC_JogSpeed");
	var[i].PlcUnitIndx = unitIU;
	var[i].unitType = unitPerc;
	var[i].DefaultUnit = UNIT_PERCENT;
	var[i].precision = 1;
	cfg->Param[i].min = 0.0;
	cfg->Param[i].max = 1.0;
	cfg->Param[i].incrMin = 0.05;
	cfg->Param[i].incrMax = 0.1;
	cfg->Param[i].defaultVal = 0.3;
	var[i].segm = 0;

	i = parOSC_MaxTvlVel;
	strcpy(var[i].name , "Max OSC Speed");
	strcpy(var[i].enumTXT, "parOSC_MaxTvlVel");
	var[i].PlcUnitIndx = unitIU;
	var[i].unitType = unitSpeed;
	var[i].DefaultUnit = UNIT_inch_per_sec;
	var[i].precision = 0;
	cfg->Param[i].min = 0.25 * in_2_mm / 1.0;
	cfg->Param[i].max = 3.0 * in_2_mm / 1.0;
	cfg->Param[i].incrMin = 0.05 * in_2_mm / 1.0;
	cfg->Param[i].incrMax = 4 * cfg->Param[i].incrMin;
	cfg->Param[i].defaultVal = 0.25 * in_2_mm / 0.5;
	var[i].segm = 0;

	//////////////////////////////////////////////////////
	//  AVC

	i = parAVC_TouchVolt;
	strcpy(var[i].name , "AVC TOUCH VOLT");
	strcpy(var[i].enumTXT, "parAVC_TouchVolt");
	var[i].PlcUnitIndx = unitIU;
	var[i].unitType = unitVolt;
	var[i].DefaultUnit = UNIT_Volt;
	var[i].precision = 1;
	cfg->Param[i].min = 0.0;
	cfg->Param[i].max = 18.0;
	cfg->Param[i].incrMin = 0.1;
	cfg->Param[i].incrMax = 1.0;
	cfg->Param[i].defaultVal = 0.6;
	var[i].segm = 0;

	i = parAVC_TouchTm;
	strcpy(var[i].name , "AVC Touch TMO");
	strcpy(var[i].enumTXT, "parAVC_TouchTm");
	var[i].PlcUnitIndx = unitIU;
	var[i].unitType = unitTime;
	var[i].DefaultUnit = UNIT_sec;
	var[i].precision = 1;
	cfg->Param[i].min = 0.0;
	cfg->Param[i].max = 60.0;
	cfg->Param[i].incrMin = 0.1;
	cfg->Param[i].incrMax = 1.0;
	cfg->Param[i].defaultVal = 5.8;
	var[i].segm = 0;

	i = parAVC_TRetractTm;
	strcpy(var[i].name , "AVC Retract Tm");
	strcpy(var[i].enumTXT, "parAVC_TRetractTm");
	var[i].PlcUnitIndx = unitIU;
	var[i].unitType = unitTime;
	var[i].DefaultUnit = UNIT_sec;
	var[i].precision = 2;
	cfg->Param[i].min = 0.0;
	cfg->Param[i].max = 10.0;
	cfg->Param[i].incrMin = 0.1;
	cfg->Param[i].incrMax = 1.0;
	cfg->Param[i].defaultVal = 0.15;
	var[i].segm = 0;

	i = parAVC_TouchRepeat;
	strcpy(var[i].name , "AVC Retry Cnt");
	strcpy(var[i].enumTXT, "parAVC_TouchRepeat");
	var[i].PlcUnitIndx = unitIU;
	var[i].unitType = unitIU;
	var[i].DefaultUnit = unitIU;
	var[i].precision = 0;
	cfg->Param[i].min = 0.0;
	cfg->Param[i].max = 10.0;
	cfg->Param[i].incrMin = 1.0;
	cfg->Param[i].incrMax = 1.0;
	cfg->Param[i].defaultVal = 3.0;
	var[i].segm = 0;

	i = parAVC_VoltInit;
	strcpy(var[i].name , "AVC INITIAL VOLT");
	strcpy(var[i].enumTXT, "parAVC_VoltInit");
	var[i].PlcUnitIndx = unitIU;
	var[i].unitType = unitVolt;
	var[i].DefaultUnit = UNIT_Volt;
	var[i].precision = 2;
	cfg->Param[i].min = 0.0;
	cfg->Param[i].max = 18.0;
	cfg->Param[i].incrMin = 0.1;
	cfg->Param[i].incrMax = 1.0;
	cfg->Param[i].defaultVal = 7.0;
	var[i].segm = 0;

	i = parAVC_VoltSP;
	strcpy(var[i].name , "PRIMARY ARC VOLTS");
	strcpy(var[i].enumTXT, "parAVC_VoltSP");
	var[i].PlcUnitIndx = unitIU;
	var[i].unitType = unitVolt;
	var[i].DefaultUnit = UNIT_Volt;
	var[i].precision = 2;
	cfg->Param[i].min = 0.0;
	cfg->Param[i].max = 30.0;
	cfg->Param[i].incrMin = 0.1;
	cfg->Param[i].incrMax = 1.0;
	cfg->Param[i].defaultVal = 10.0;
	var[i].segm = 1;

	i = parAVC_VoltInSP;
	strcpy(var[i].name , "PRIMARY In ARC VOLTS");
	strcpy(var[i].enumTXT, "parAVC_VoltInSP");
	var[i].PlcUnitIndx = unitIU;
	var[i].unitType = unitVolt;
	var[i].DefaultUnit = UNIT_Volt;
	var[i].precision = 2;
	cfg->Param[i].min = 0.0;
	cfg->Param[i].max = 30.0;
	cfg->Param[i].incrMin = 0.1;
	cfg->Param[i].incrMax = 1.0;
	cfg->Param[i].defaultVal = 10.0;
	var[i].segm = 1;

	i = parAVC_VoltOutSP;
	strcpy(var[i].name , "PRIMARY Out ARC VOLTS");
	strcpy(var[i].enumTXT, "parAVC_VoltOutSP");
	var[i].PlcUnitIndx = unitIU;
	var[i].unitType = unitVolt;
	var[i].DefaultUnit = UNIT_Volt;
	var[i].precision = 2;
	cfg->Param[i].min = 0.0;
	cfg->Param[i].max = 30.0;
	cfg->Param[i].incrMin = 0.1;
	cfg->Param[i].incrMax = 1.0;
	cfg->Param[i].defaultVal = 10.0;
	var[i].segm = 1;

	 i = parAVC_VoltBackSP;
	strcpy(var[i].name , "BACKGRD ARC VOLTS");
	strcpy(var[i].enumTXT, "parAVC_VoltBackSP");
	var[i].PlcUnitIndx = unitIU;
	var[i].unitType = unitVolt;
	var[i].DefaultUnit = UNIT_Volt;
	var[i].precision = 2;
	cfg->Param[i].min = 0.0;
	cfg->Param[i].max = 30.0;
	cfg->Param[i].incrMin = 0.1;
	cfg->Param[i].incrMax = 1.0;
	cfg->Param[i].defaultVal = 10.0;
	var[i].segm = 1;

	i = parAVC_Boost1;
	strcpy(var[i].name , "Boost1 ARC VOLTS");
	strcpy(var[i].enumTXT, "parAVC_Boost1");
	var[i].PlcUnitIndx = unitIU;
	var[i].unitType = unitVolt;
	var[i].DefaultUnit = UNIT_Volt;
	var[i].precision = 2;
	cfg->Param[i].max = 30.0;
	cfg->Param[i].min = -cfg->Param[i].max;
	cfg->Param[i].incrMin = 0.1;
	cfg->Param[i].incrMax = 1.0;
	cfg->Param[i].defaultVal = 0.0;
	var[i].segm = 1;

	i = parAVC_Boost2;
	strcpy(var[i].name , "Boost2 ARC VOLTS");
	strcpy(var[i].enumTXT, "parAVC_Boost2");
	var[i].PlcUnitIndx = unitIU;
	var[i].unitType = unitVolt;
	var[i].DefaultUnit = UNIT_Volt;
	var[i].precision = 2;
	cfg->Param[i].max = 30.0;
	cfg->Param[i].min = -cfg->Param[i].max;
	cfg->Param[i].incrMin = 0.1;
	cfg->Param[i].incrMax = 1.0;
	cfg->Param[i].defaultVal = 0.0;
	var[i].segm = 1;

	i = parAVC_VSPTmOut;
	strcpy(var[i].name , "AVC Prim Volt Tmo");
	strcpy(var[i].enumTXT, "parAVC_VSPTmOut");
	var[i].PlcUnitIndx = unitIU;
	var[i].unitType = unitTime;
	var[i].DefaultUnit = UNIT_sec;
	var[i].precision = 1;
	cfg->Param[i].min = 0.0;
	cfg->Param[i].max = 10.0;
	cfg->Param[i].incrMin = 0.1;
	cfg->Param[i].incrMax = 1.0;
	cfg->Param[i].defaultVal = 10;
	var[i].segm = 0;

	i = parAVC_TouchVel;
	strcpy(var[i].name , "AVC SLOW RUN IN SP");
	strcpy(var[i].enumTXT, "parAVC_TouchVel");
	var[i].PlcUnitIndx = unitIU;
	var[i].unitType = unitPerc;
	var[i].DefaultUnit = UNIT_PERCENT;
	var[i].precision = 1;
	cfg->Param[i].min = 0.0;
	cfg->Param[i].max = 1.0;
	cfg->Param[i].incrMin = 0.05;
	cfg->Param[i].incrMax = 0.1;
	cfg->Param[i].defaultVal = 0.15;
	var[i].segm = 0;

	i = parAVC_ToSPVel;
	strcpy(var[i].name , "AVC LIFT UP SPEED");
	strcpy(var[i].enumTXT, "parAVC_ToSPVel");
	var[i].PlcUnitIndx = unitIU;
	var[i].unitType = unitPerc;
	var[i].DefaultUnit = UNIT_PERCENT;
	var[i].precision = 1;
	cfg->Param[i].min = 0.0;
	cfg->Param[i].max = 1.0;
	cfg->Param[i].incrMin = 0.05;
	cfg->Param[i].incrMax = 0.1;
	cfg->Param[i].defaultVal = 0.5;
	var[i].segm = 0;

	i = parAVC_LU_TM;
	strcpy(var[i].name , "AVC LU TM");
	strcpy(var[i].enumTXT, "parAVC_LU_TM");
	var[i].PlcUnitIndx = unitIU;
	var[i].unitType = unitTime;
	var[i].DefaultUnit = UNIT_sec;
	var[i].precision = 2;
	cfg->Param[i].min = 0.01;
	cfg->Param[i].max = 2.0;
	cfg->Param[i].incrMin = 0.01;
	cfg->Param[i].incrMax = 0.1;
	cfg->Param[i].defaultVal = 0.2;
	var[i].segm = 0;

	i = parAVC_KissTm;
	strcpy(var[i].name , "AVC Kiss TM");
	strcpy(var[i].enumTXT, "parAVC_KissTm");
	var[i].PlcUnitIndx = unitIU;
	var[i].unitType = unitTime;
	var[i].DefaultUnit = UNIT_sec;
	var[i].precision = 2;
	cfg->Param[i].min = 0.005;
	cfg->Param[i].max = 2.0;
	cfg->Param[i].incrMin = 0.005;
	cfg->Param[i].incrMax = 0.1;
	cfg->Param[i].defaultVal = 0.01;
	var[i].segm = 0;

	i = parAVC_Upslope;
	strcpy(var[i].name , "VOLT UPSLOPE TM");
	strcpy(var[i].enumTXT, "parAVC_Upslope");
	var[i].PlcUnitIndx = unitIU;
	var[i].unitType = unitTime;
	var[i].DefaultUnit = UNIT_sec;
	var[i].precision = 1;
	cfg->Param[i].min = 0.0;
	cfg->Param[i].max = 30.0;
	cfg->Param[i].incrMin = 0.1;
	cfg->Param[i].incrMax = 1.0;
	cfg->Param[i].defaultVal = 3.0;
	var[i].segm = 0;

	i = parAVC_DownSlope;
	strcpy(var[i].name , "VOLT DOWNSLOPE TM");
	strcpy(var[i].enumTXT, "parAVC_DownSlope");
	var[i].PlcUnitIndx = unitIU;
	var[i].unitType = unitTime;
	var[i].DefaultUnit = UNIT_sec;
	var[i].precision = 1;
	cfg->Param[i].min = 0.0;
	cfg->Param[i].max = 20.0;
	cfg->Param[i].incrMin = 0.1;
	cfg->Param[i].incrMax = 1.0;
	cfg->Param[i].defaultVal = 1.0;
	var[i].segm = 0;

	i = parAVC_HoldTm;
	strcpy(var[i].name , "AVC RETRACT DLY");
	strcpy(var[i].enumTXT, "parAVC_HoldTm");
	var[i].PlcUnitIndx = unitIU;
	var[i].unitType = unitTime;
	var[i].DefaultUnit = UNIT_sec;
	var[i].precision = 1;
	cfg->Param[i].min = 0.0;
	cfg->Param[i].max = 60.0;
	cfg->Param[i].incrMin = 0.1;
	cfg->Param[i].incrMax = 1.0;
	cfg->Param[i].defaultVal = 10.0;
	var[i].segm = 0;

	i = parAVC_VoltFinal;
	strcpy(var[i].name , "FINAL ARC VOLTS");
	strcpy(var[i].enumTXT, "parAVC_VoltFinal");
	var[i].PlcUnitIndx = unitIU;
	var[i].unitType = unitVolt;
	var[i].DefaultUnit = UNIT_Volt;
	var[i].precision = 2;
	cfg->Param[i].min = 0.0;
	cfg->Param[i].max = 18.0;
	cfg->Param[i].incrMin = 0.1;
	cfg->Param[i].incrMax = 1.0;
	cfg->Param[i].defaultVal = 9.0;
	var[i].segm = 0;

	i = parAVC_GoBackTm;
	strcpy(var[i].name , "AVC RETRACT TM");
	strcpy(var[i].enumTXT, "parAVC_GoBackTm");
	var[i].PlcUnitIndx = unitIU;
	var[i].unitType = unitTime;
	var[i].DefaultUnit = UNIT_sec;
	var[i].precision = 1;
	cfg->Param[i].min = 0.0;
	cfg->Param[i].max = 5.0;
	cfg->Param[i].incrMin = 0.1;
	cfg->Param[i].incrMax = 1.0;
	cfg->Param[i].defaultVal = 2.0;
	var[i].segm = 0;

	i = parAVC_StartDly;
	strcpy(var[i].name , "VOLT UPSLOPE DLY");
	strcpy(var[i].enumTXT, "parAVC_StartDly");
	var[i].PlcUnitIndx = unitIU;
	var[i].unitType = unitTime;
	var[i].DefaultUnit = UNIT_sec;
	var[i].precision = 1;
	cfg->Param[i].min = 0.0;
	cfg->Param[i].max = 10.0;
	cfg->Param[i].incrMin = 0.1;
	cfg->Param[i].incrMax = 1.0;
	cfg->Param[i].defaultVal = 2.0;
	var[i].segm = 0;

	i = parAVC_StopDly;
	strcpy(var[i].name , "VOLT DWNSLOPE DLY");
	strcpy(var[i].enumTXT, "parAVC_StopDly");
	var[i].PlcUnitIndx = unitIU;
	var[i].unitType = unitTime;
	var[i].DefaultUnit = UNIT_sec;
	var[i].precision = 1;
	cfg->Param[i].min = 0.0;
	cfg->Param[i].max = 10.0;
	cfg->Param[i].incrMin = 0.1;
	cfg->Param[i].incrMax = 1.0;
	cfg->Param[i].defaultVal = 1.0;
	var[i].segm = 0;

	i = parAVC_MaxVoltError;
	strcpy(var[i].name , "AVC Max Volt Err");
	strcpy(var[i].enumTXT, "parAVC_MaxVoltError");
	var[i].PlcUnitIndx = unitIU;
	var[i].unitType = unitVolt;
	var[i].DefaultUnit = UNIT_Volt;
	var[i].precision = 2;
	cfg->Param[i].min = 0.0;
	cfg->Param[i].max = 10.0;
	cfg->Param[i].incrMin = 0.1;
	cfg->Param[i].incrMax = 1.0;
	cfg->Param[i].defaultVal = 10.0;
	var[i].segm = 0;

	i = parAVC_Limits_Mask_Tm;
	strcpy(var[i].name , "AVC Limits Filter Tm");
	strcpy(var[i].enumTXT, "parAVC_Limits_Mask_Tm");
	var[i].PlcUnitIndx = unitIU;
	var[i].unitType = unitTime;
	var[i].DefaultUnit = UNIT_sec;
	var[i].precision = 3;
	cfg->Param[i].min = 0.0;
	cfg->Param[i].max = 2.0;
	cfg->Param[i].incrMin = 0.05;
	cfg->Param[i].incrMax = 0.2;
	cfg->Param[i].defaultVal = 0.1;
	var[i].segm = 0;

	i = parAVC_JogSpeedDirCntrl;
	strcpy(var[i].name , "AVC Jog Speed");
	strcpy(var[i].enumTXT, "parAVC_JogSpeedDirCntrl");
	var[i].PlcUnitIndx = unitIU;
	var[i].unitType = unitPerc;
	var[i].DefaultUnit = UNIT_PERCENT;
	var[i].precision = 1;
	cfg->Param[i].min = 0.0;
	cfg->Param[i].max = 1.0;
	cfg->Param[i].incrMin = 0.05;
	cfg->Param[i].incrMax = 0.1;
	cfg->Param[i].defaultVal = 0.75;
	var[i].segm = 0;

	i = parAVC_LiftSpeedDirCntrl;
	strcpy(var[i].name , "AVC RETRACT SP");
	strcpy(var[i].enumTXT, "parAVC_LiftSpeedDirCntrl");
	var[i].PlcUnitIndx = unitIU;
	var[i].unitType = unitPerc;
	var[i].DefaultUnit = UNIT_PERCENT;
	var[i].precision = 1;
	cfg->Param[i].min = 0.0;
	cfg->Param[i].max = 1.0;
	cfg->Param[i].incrMin = 0.05;
	cfg->Param[i].incrMax = 0.1;
	cfg->Param[i].defaultVal = 0.35;
	var[i].segm = 0;

	i = parAVC_FbkFilter;
	strcpy(var[i].name , "AVC Sign Filter");
	strcpy(var[i].enumTXT, "parAVC_FbkFilter");
	var[i].PlcUnitIndx = unitIU;
	var[i].unitType = unitPerc;
	var[i].DefaultUnit = UNIT_PERCENT;
	var[i].precision = 1;
	cfg->Param[i].min = 0.0;
	cfg->Param[i].max = 1.0;
	cfg->Param[i].incrMin = 0.01;
	cfg->Param[i].incrMax = 0.1;
	cfg->Param[i].defaultVal = 0.0;
	var[i].segm = 0;

	i = parAVC_KPP;
	strcpy(var[i].name , "AVC KPP");
	strcpy(var[i].enumTXT, "parAVC_KPP");
	var[i].PlcUnitIndx = unitIU;
	var[i].unitType = unitPerc;
	var[i].DefaultUnit = UNIT_PERCENT;
	var[i].precision = 1;
	cfg->Param[i].min = 0.0;
	cfg->Param[i].max = 1.0;
	cfg->Param[i].incrMin = 0.01;
	cfg->Param[i].incrMax = 0.1;
	cfg->Param[i].defaultVal = 0.5;
	var[i].segm = 0;

	i = parAVC_KIP;
	strcpy(var[i].name , "AVC KIP");
	strcpy(var[i].enumTXT, "parAVC_KIP");
	var[i].PlcUnitIndx = unitIU;
	var[i].unitType = unitPerc;
	var[i].DefaultUnit = UNIT_PERCENT;
	var[i].precision = 1;
	cfg->Param[i].min = 0.0;
	cfg->Param[i].max = 1.0;
	cfg->Param[i].incrMin = 0.01;
	cfg->Param[i].incrMax = 0.1;
	cfg->Param[i].defaultVal = 0.1;
	var[i].segm = 0;

	i = parAVC_BB_Vel;
	strcpy(var[i].name , "AVC BB Speed");
	strcpy(var[i].enumTXT, "parAVC_BB_Vel");
	var[i].PlcUnitIndx = unitIU;
	var[i].unitType = unitPerc;
	var[i].DefaultUnit = UNIT_PERCENT;
	var[i].precision = 1;
	cfg->Param[i].min = 0.0;
	cfg->Param[i].max = 1.0;
	cfg->Param[i].incrMin = 0.01;
	cfg->Param[i].incrMax = 0.1;
	cfg->Param[i].defaultVal = 0.15;
	var[i].segm = 0;

	i = parAVC_BB_Integr;
	strcpy(var[i].name , "AVC BB Integr");
	strcpy(var[i].enumTXT, "parAVC_BB_Integr");
	var[i].PlcUnitIndx = unitIU;
	var[i].unitType = unitPerc;
	var[i].DefaultUnit = UNIT_PERCENT;
	var[i].precision = 2;
	cfg->Param[i].min = 0.0;
	cfg->Param[i].max = 1.0;
	cfg->Param[i].incrMin = 0.01;
	cfg->Param[i].incrMax = 0.1;
	cfg->Param[i].defaultVal = 0.25;
	var[i].segm = 0;

	i = parAVC_BB_Gain;
	strcpy(var[i].name , "AVC BB Gain");
	strcpy(var[i].enumTXT, "parAVC_BB_Gain");
	var[i].PlcUnitIndx = unitIU;
	var[i].unitType = unitIU;
	var[i].DefaultUnit = unitIU;
	var[i].precision = 1;
	cfg->Param[i].min = 0.0;
	cfg->Param[i].max = 10.0;
	cfg->Param[i].incrMin = 0.01;
	cfg->Param[i].incrMax = 0.1;
	cfg->Param[i].defaultVal = 0.5;
	var[i].segm = 0;

	i = parAVC_DB_Window;
	strcpy(var[i].name , "AVC DB Window");
	strcpy(var[i].enumTXT, "parAVC_DB_Window");
	var[i].PlcUnitIndx = unitIU;
	var[i].unitType = unitVolt;
	var[i].DefaultUnit = UNIT_Volt;
	var[i].precision = 2;
	cfg->Param[i].min = 0.0;
	cfg->Param[i].max = 2.0;
	cfg->Param[i].incrMin = 0.01;
	cfg->Param[i].incrMax = 0.5;
	cfg->Param[i].defaultVal = 0.3;
	var[i].segm = 0;

	//////////////////////////////////////////////////////
	//  Wire Feed
	i = parWF_StartDly;
	strcpy(var[i].name , "WF START DLY");
	strcpy(var[i].enumTXT, "parWF_StartDly");
	var[i].PlcUnitIndx = unitIU;
	var[i].unitType = unitTime;
	var[i].DefaultUnit = UNIT_sec;
	var[i].precision = 1;
	cfg->Param[i].min = 0.0;
	cfg->Param[i].max = 60.0;
	cfg->Param[i].incrMin = 0.1;
	cfg->Param[i].incrMax = 1.0;
	cfg->Param[i].defaultVal = 5.0;
	var[i].segm = 0;

	i = parWF_RampUp;
	strcpy(var[i].name , "WF UPSLOPE TM");
	strcpy(var[i].enumTXT, "parWF_RampUp");
	var[i].PlcUnitIndx = unitIU;
	var[i].unitType = unitTime;
	var[i].DefaultUnit = UNIT_sec;
	var[i].precision = 1;
	cfg->Param[i].min = 0.0;
	cfg->Param[i].max = 60.0;
	cfg->Param[i].incrMin = 0.1;
	cfg->Param[i].incrMax = 1.0;
	cfg->Param[i].defaultVal = 4.0;
	var[i].segm = 0;

	i = parWF_SpeedSP;
	strcpy(var[i].name , "WF PRIMARY SPEED");
	strcpy(var[i].enumTXT, "parWF_SpeedSP");
	var[i].PlcUnitIndx = unitIU;
	var[i].unitType = unitSpeed;
	var[i].DefaultUnit = UNIT_inch_per_min;
	var[i].precision = 0;
	cfg->Param[i].max = 500 * in_min_2_mm_s;
	cfg->Param[i].incrMin = 1 * in_min_2_mm_s;
	cfg->Param[i].incrMax = 10.0 * cfg->Param[i].incrMin;
	cfg->Param[i].defaultVal = 100.0 * in_min_2_mm_s;
	var[i].segm = 1;

	i = parWF_SpeedInSP;
	strcpy(var[i].name , "WF PRIMARY IN SPEED");
	strcpy(var[i].enumTXT, "parWF_SpeedInSP");
	var[i].PlcUnitIndx = unitIU;
	var[i].unitType = unitSpeed;
	var[i].DefaultUnit = UNIT_inch_per_min;
	var[i].precision = 0;
	cfg->Param[i].max = 500 * in_min_2_mm_s;
	cfg->Param[i].incrMin = 1 * in_min_2_mm_s;
	cfg->Param[i].incrMax = 10.0 * cfg->Param[i].incrMin;
	cfg->Param[i].defaultVal = 100.0 * in_min_2_mm_s;
	var[i].segm = 1;

	i = parWF_SpeedOutSP;
	strcpy(var[i].name , "WF PRIMARY OUT SPEED");
	strcpy(var[i].enumTXT, "parWF_SpeedOutSP");
	var[i].PlcUnitIndx = unitIU;
	var[i].unitType = unitSpeed;
	var[i].DefaultUnit = UNIT_inch_per_min;
	var[i].precision = 0;
	cfg->Param[i].max = 500 * in_min_2_mm_s;
	cfg->Param[i].incrMin = 1 * in_min_2_mm_s;
	cfg->Param[i].incrMax = 10.0 * cfg->Param[i].incrMin;
	cfg->Param[i].defaultVal = 100.0 * in_min_2_mm_s;
	var[i].segm = 1;

	i = parWF_BkgSpeedSP;
	strcpy(var[i].name , "WF BKG SPEED");
	strcpy(var[i].enumTXT, "parWF_BkgSpeedSP");
	var[i].PlcUnitIndx = unitIU;
	var[i].unitType = unitSpeed;
	var[i].DefaultUnit = UNIT_inch_per_min;
	var[i].precision = 0;
	cfg->Param[i].max = 500 * in_min_2_mm_s;
	cfg->Param[i].incrMin = 1 * in_min_2_mm_s;
	cfg->Param[i].incrMax = 10.0 * cfg->Param[i].incrMin;
	cfg->Param[i].defaultVal = 100.0 * in_min_2_mm_s;
	var[i].segm = 1;

	i = parWF_SpeedInit;
	strcpy(var[i].name , "WF INITIAL SPEED");
	strcpy(var[i].enumTXT, "parWF_SpeedInit");
	var[i].PlcUnitIndx = unitIU;
	var[i].unitType = unitSpeed;
	var[i].DefaultUnit = UNIT_inch_per_min;
	var[i].precision = 0;
	cfg->Param[i].max = 100.0;
	cfg->Param[i].incrMin = 1 * in_min_2_mm_s;
	cfg->Param[i].incrMax = 10.0 * cfg->Param[i].incrMin;
	cfg->Param[i].defaultVal =0.0 * in_min_2_mm_s;
	var[i].segm = 0;

	i = parWF_SpeedFinal;
	strcpy(var[i].name , "WF FINAL SPEED");
	strcpy(var[i].enumTXT, "parWF_SpeedFinal");
	var[i].PlcUnitIndx = unitIU;
	var[i].unitType = unitSpeed;
	var[i].DefaultUnit = UNIT_inch_per_min;
	var[i].precision = 0;
	cfg->Param[i].max = 100.0;
	cfg->Param[i].incrMin = 1 * in_min_2_mm_s;
	cfg->Param[i].incrMax = 10.0 * cfg->Param[i].incrMin;
	cfg->Param[i].defaultVal = 0.0 * in_min_2_mm_s;
	var[i].segm = 0;

	i = parWF_StopDly;
	strcpy(var[i].name , "WF DOWNSLOPE DLY");
	strcpy(var[i].enumTXT, "parWF_StopDly");
	var[i].PlcUnitIndx = unitIU;
	var[i].unitType = unitTime;
	var[i].DefaultUnit = UNIT_sec;
	var[i].precision = 1;
	cfg->Param[i].min = 0.0;
	cfg->Param[i].max = 60.0;
	cfg->Param[i].incrMin = 0.1;
	cfg->Param[i].incrMax = 1.0;
	cfg->Param[i].defaultVal = 2.0;
	var[i].segm = 0;

	i = parWF_RampDwn;
	strcpy(var[i].name , "WF DOWNSLOPE TIME");
	strcpy(var[i].enumTXT, "parWF_RampDwn");
	var[i].PlcUnitIndx = unitIU;
	var[i].unitType = unitTime;
	var[i].DefaultUnit = UNIT_sec;
	var[i].precision = 1;
	cfg->Param[i].min = 0.0;
	cfg->Param[i].max = 60.0;
	cfg->Param[i].incrMin = 0.1;
	cfg->Param[i].incrMax = 1.0;
	cfg->Param[i].defaultVal = 0.5;
	var[i].segm = 0;

	i = parWF_RampUpdate;
	strcpy(var[i].name , "WF Ramp Update");
	strcpy(var[i].enumTXT, "parWF_RampUpdate");
	var[i].PlcUnitIndx = unitIU;
	var[i].unitType = unitTime;
	var[i].DefaultUnit = UNIT_sec;
	var[i].precision = 1;
	cfg->Param[i].min = 0.0;
	cfg->Param[i].max = 60.0;
	cfg->Param[i].incrMin = 0.1;
	cfg->Param[i].incrMax = 1.0;
	cfg->Param[i].defaultVal = 0.1;

	i = parWF_Boost1SP;
	strcpy(var[i].name , "WF Boost1");
	strcpy(var[i].enumTXT, "parWF_Boost1SP");
	var[i].PlcUnitIndx = unitIU;
	var[i].unitType = unitSpeed;
	var[i].DefaultUnit = UNIT_inch_per_min;
	var[i].precision = 0;
	cfg->Param[i].max = 500 * in_min_2_mm_s;
	cfg->Param[i].min = -cfg->Param[i].max;
	cfg->Param[i].incrMin = 1 * in_min_2_mm_s;
	cfg->Param[i].incrMax = 10.0 * cfg->Param[i].incrMin;
	cfg->Param[i].defaultVal = 0.0;
	var[i].segm = 1;

	i = parWF_Boost2SP;
	strcpy(var[i].name , "WF Boots2");
	strcpy(var[i].enumTXT, "parWF_Boost2SP");
	var[i].PlcUnitIndx = unitIU;
	var[i].unitType = unitSpeed;
	var[i].DefaultUnit = UNIT_inch_per_min;
	var[i].precision = 0;
	cfg->Param[i].max = 500 * in_min_2_mm_s;
	cfg->Param[i].min = -cfg->Param[i].max;
	cfg->Param[i].incrMin = 1 * in_min_2_mm_s;
	cfg->Param[i].incrMax = 10.0 * cfg->Param[i].incrMin;
	cfg->Param[i].defaultVal = 0.0;
	var[i].segm = 1;

	 i = parWF_JogSpeed;
	strcpy(var[i].name , "WF Jog ???");
	strcpy(var[i].enumTXT, "parWF_JogSpeed");
	var[i].PlcUnitIndx = unitIU;
	var[i].unitType = unitPerc;
	var[i].DefaultUnit = UNIT_PERCENT;
	var[i].precision = 0;
	cfg->Param[i].min = 0.0;
	cfg->Param[i].max = 1.0;
	cfg->Param[i].incrMin = 0.01;
	cfg->Param[i].incrMax = 0.1;
	cfg->Param[i].defaultVal = 0.5;
	var[i].segm = 0;

	i = parWF_JogSpeedDirCntrl;
	strcpy(var[i].name , "WF Jog Speed");
	strcpy(var[i].enumTXT, "parWF_JogSpeedDirCntrl");
	var[i].PlcUnitIndx = unitIU;
	var[i].unitType = unitPerc;
	var[i].DefaultUnit = UNIT_PERCENT;
	var[i].precision = 0;
	cfg->Param[i].min = 0.0;
	cfg->Param[i].max = 1.0;
	cfg->Param[i].incrMin = 0.01;
	cfg->Param[i].incrMax = 0.1;
	cfg->Param[i].defaultVal = 0.9;
	var[i].segm = 0;

	i = parWF_RetractDly;
	strcpy(var[i].name , "WF RETRACT DLY");
	strcpy(var[i].enumTXT, "parWF_RetractDly");
	var[i].PlcUnitIndx = unitIU;
	var[i].unitType = unitTime;
	var[i].DefaultUnit = UNIT_sec;
	var[i].precision = 1;
	cfg->Param[i].min = 0.0;
	cfg->Param[i].max = 120.0;
	cfg->Param[i].incrMin = 0.1;
	cfg->Param[i].incrMax = 1.0;
	cfg->Param[i].defaultVal = 9.0;
	var[i].segm = 0;

	i = parWF_RetractSpeed;
	strcpy(var[i].name , "WF RETRACT SPEED");
	strcpy(var[i].enumTXT, "parWF_RetractSpeed");
	var[i].PlcUnitIndx = unitIU;
	var[i].unitType = unitPerc;
	var[i].DefaultUnit = UNIT_PERCENT;
	var[i].precision = 1;
	cfg->Param[i].min = 0.0;
	cfg->Param[i].max = 1.0;
	cfg->Param[i].incrMin = 0.05;
	cfg->Param[i].incrMax = 0.1;
	cfg->Param[i].defaultVal = 0.25;
	var[i].segm = 0;

	i = parWF_RetracDist;
	strcpy(var[i].name , "WF RETRACT LENGTH");
	strcpy(var[i].enumTXT, "parWF_RetracDist");
	var[i].PlcUnitIndx = unitIU;
	var[i].unitType = unitLength;
	var[i].DefaultUnit = UNIT_inch;
	var[i].precision = 1;
	cfg->Param[i].min = 0.0;
	cfg->Param[i].max = 25.4 * 2;
	cfg->Param[i].incrMin = 0.1;
	cfg->Param[i].incrMax = 1.0;
	cfg->Param[i].defaultVal = 0.2 * in_2_mm;
	var[i].segm = 0;

	i = parWF_CalibVel1;
	strcpy(var[i].name , "WF Calib Speed 1");
	strcpy(var[i].enumTXT, "parWF_CalibVel1");
	var[i].PlcUnitIndx = unitIU;
	var[i].unitType = unitSpeed;
	var[i].DefaultUnit = UNIT_inch_per_min;
	var[i].precision = 0;
	cfg->Param[i].max = 127.0;
	cfg->Param[i].incrMin = 1 * in_min_2_mm_s;
	cfg->Param[i].incrMax = 10.0 * cfg->Param[i].incrMin;
	cfg->Param[i].defaultVal = 50.0 * in_min_2_mm_s;
	var[i].segm = 0;

	i = parWF_CalibVel2;
	strcpy(var[i].name , "WF Calib Speed 2");
	strcpy(var[i].enumTXT, "parWF_CalibVel2");
	var[i].PlcUnitIndx = unitIU;
	var[i].unitType = unitSpeed;
	var[i].DefaultUnit = UNIT_inch_per_min;
	var[i].precision = 0;
	cfg->Param[i].max = 127.0;
	cfg->Param[i].incrMin = 1 * in_min_2_mm_s;
	cfg->Param[i].incrMax = 10.0 * cfg->Param[i].incrMin;
	cfg->Param[i].defaultVal = 100.0 * in_min_2_mm_s;
	var[i].segm = 0;

	//////////////////////////////////////////////////////
	//	Wire Pulse

	i = parWP_StartDly;
	strcpy(var[i].name , "WP START DELAY");
	strcpy(var[i].enumTXT, "parWP_StartDly");
	var[i].PlcUnitIndx = unitIU;
	var[i].unitType = unitTime;
	var[i].DefaultUnit = UNIT_sec;
	var[i].precision = 1;
	cfg->Param[i].min = 0.0;
	cfg->Param[i].max = 60.0;
	cfg->Param[i].incrMin = 0.1;
	cfg->Param[i].incrMax = 1.0;
	cfg->Param[i].defaultVal = 5.0;
	var[i].segm = 0;

	i = parWP_RampUp;
	strcpy(var[i].name , "WP UPSLOPE TM");
	strcpy(var[i].enumTXT, "parWP_RampUp");
	var[i].PlcUnitIndx = unitIU;
	var[i].unitType = unitTime;
	var[i].DefaultUnit = UNIT_sec;
	var[i].precision = 1;
	cfg->Param[i].min = 0.0;
	cfg->Param[i].max = 60.0;
	cfg->Param[i].incrMin = 0.1;
	cfg->Param[i].incrMax = 1.0;
	cfg->Param[i].defaultVal = 3.0;
	var[i].segm = 0;

	i = parWP_SpeedSP;
	strcpy(var[i].name , "WP PRIMARY SPEED");
	strcpy(var[i].enumTXT, "parWP_SpeedSP");
	var[i].PlcUnitIndx = unitIU;
	var[i].unitType = unitFreq;
	var[i].DefaultUnit = UNIT_Hz;
	var[i].precision = 1;
	cfg->Param[i].max = 40.0;
	cfg->Param[i].incrMin = 0.1;
	cfg->Param[i].incrMax = 1.0;
	cfg->Param[i].defaultVal = 13.2;
	var[i].segm = 1;

	i = parWP_SpeedInSP;
	strcpy(var[i].name , "WP PRIMARY IN SPEED");
	strcpy(var[i].enumTXT, "parWP_SpeedInSP");
	var[i].PlcUnitIndx = unitIU;
	var[i].unitType = unitFreq;
	var[i].DefaultUnit = UNIT_Hz;
	var[i].precision = 1;
	cfg->Param[i].max = 40.0;
	cfg->Param[i].incrMin = 0.1;
	cfg->Param[i].incrMax = 1.0;
	cfg->Param[i].defaultVal = 13.2;
	var[i].segm = 1;

	i = parWP_SpeedOutSP;
	strcpy(var[i].name , "WP PRIMARY OUT SPEED");
	strcpy(var[i].enumTXT, "parWP_SpeedOutSP");
	var[i].PlcUnitIndx = unitIU;
	var[i].unitType = unitFreq;
	var[i].DefaultUnit = UNIT_Hz;
	var[i].precision = 1;
	cfg->Param[i].max = 40.0;
	cfg->Param[i].incrMin = 0.1;
	cfg->Param[i].incrMax = 1.0;
	cfg->Param[i].defaultVal = 13.2;
	var[i].segm = 1;

	i = parWP_BkgSpeedSP;
	strcpy(var[i].name , "WP BKG SPEED");
	strcpy(var[i].enumTXT, "parWP_BkgSpeedSP");
	var[i].PlcUnitIndx = unitIU;
	var[i].unitType = unitFreq;
	var[i].DefaultUnit = UNIT_Hz;
	var[i].precision = 1;
	cfg->Param[i].max = 40.0;
	cfg->Param[i].incrMin = 0.1;
	cfg->Param[i].incrMax = 1.0;
	cfg->Param[i].defaultVal = 13.2;
	var[i].segm = 1;

	i = parWP_SpeedInit;
	strcpy(var[i].name , "WP INITIAL SPEED");
	strcpy(var[i].enumTXT, "parWP_SpeedInit");
	var[i].PlcUnitIndx = unitIU;
	var[i].unitType = unitFreq;
	var[i].DefaultUnit = UNIT_Hz;
	var[i].precision = 1;
	cfg->Param[i].max = 25.0;
	cfg->Param[i].incrMin = 0.25;
	cfg->Param[i].incrMax = 1.0;
	cfg->Param[i].defaultVal = 0.0;
	var[i].segm = 0;

	i = parWP_SpeedFinal;
	strcpy(var[i].name , "WP FINAL SPEED");
	strcpy(var[i].enumTXT, "parWP_SpeedFinal");
	var[i].PlcUnitIndx = unitIU;
	var[i].unitType = unitFreq;
	var[i].DefaultUnit = UNIT_Hz;
	var[i].precision = 1;
	cfg->Param[i].max = 25.0;
	cfg->Param[i].incrMin = 0.25;
	cfg->Param[i].incrMax = 1.0;
	cfg->Param[i].defaultVal = 0.0;
	var[i].segm = 0;

	i = parWP_StopDly;
	strcpy(var[i].name , "WP DOWNSLOPE DLY");
	strcpy(var[i].enumTXT, "parWP_StopDly");
	var[i].PlcUnitIndx = unitIU;
	var[i].unitType = unitTime;
	var[i].DefaultUnit = UNIT_sec;
	var[i].precision = 1;
	cfg->Param[i].min = 0.0;
	cfg->Param[i].max = 60.0;
	cfg->Param[i].incrMin = 0.1;
	cfg->Param[i].incrMax = 1.0;
	cfg->Param[i].defaultVal = 2.0;
	var[i].segm = 0;

	i = parWP_RampDwn;
	strcpy(var[i].name , "WP DOWNSLOPE TM");
	strcpy(var[i].enumTXT, "parWP_RampDwn");
	var[i].PlcUnitIndx = unitIU;
	var[i].unitType = unitTime;
	var[i].DefaultUnit = UNIT_sec;
	var[i].precision = 1;
	cfg->Param[i].min = 0.0;
	cfg->Param[i].max = 60.0;
	cfg->Param[i].incrMin = 0.1;
	cfg->Param[i].incrMax = 1.0;
	cfg->Param[i].defaultVal = 0.5;
	var[i].segm = 0;

	i = parWP_RampUpdate;
	strcpy(var[i].name , "WP Ramp Update");
	strcpy(var[i].enumTXT, "parWP_RampUpdate");
	var[i].PlcUnitIndx = unitIU;
	var[i].unitType = unitTime;
	var[i].DefaultUnit = UNIT_sec;
	var[i].precision = 1;
	cfg->Param[i].min = 0.0;
	cfg->Param[i].max = 60.0;
	cfg->Param[i].incrMin = 0.1;
	cfg->Param[i].incrMax = 1.0;
	cfg->Param[i].defaultVal = 0.1;
	var[i].segm = 0;

	i = parWP_Boost1SP;
	strcpy(var[i].name , "WP Boot1");
	strcpy(var[i].enumTXT, "parWP_Boost1SP");
	var[i].PlcUnitIndx = unitIU;
	var[i].unitType = unitFreq;
	var[i].DefaultUnit = UNIT_Hz;
	var[i].precision = 1;
	cfg->Param[i].max = 40.0;
	cfg->Param[i].min = -cfg->Param[i].max;
	cfg->Param[i].incrMin = 0.1;
	cfg->Param[i].incrMax = 1.0;
	cfg->Param[i].defaultVal = 0.0;
	var[i].segm = 1;

	i = parWP_Boost2SP;
	strcpy(var[i].name , "WP Boot2");
	strcpy(var[i].enumTXT, "parWP_Boost2SP");
	var[i].PlcUnitIndx = unitIU;
	var[i].unitType = unitFreq;
	var[i].DefaultUnit = UNIT_Hz;
	var[i].precision = 1;
	cfg->Param[i].max = 40.0;
	cfg->Param[i].min = -cfg->Param[i].max;
	cfg->Param[i].incrMin = 0.1;
	cfg->Param[i].incrMax = 1.0;
	cfg->Param[i].defaultVal = 0.0;
	var[i].segm = 1;

	i = parWP_JogSpeed;
	strcpy(var[i].name , "WP Jog");
	strcpy(var[i].enumTXT, "parWP_JogSpeed");
	var[i].PlcUnitIndx = unitIU;
	var[i].unitType = unitFreq;
	var[i].DefaultUnit = UNIT_Hz;
	var[i].precision = 1;
	cfg->Param[i].max = 25.0;
	cfg->Param[i].incrMin = 0.25;
	cfg->Param[i].incrMax = 1.0;
	cfg->Param[i].defaultVal = 6.0;
	var[i].segm = 0;

	i = parWP_JogSpeedDirCntrl;
	strcpy(var[i].name , "WP Jog Cntrl");
	strcpy(var[i].enumTXT, "parWP_JogSpeedDirCntrl");
	var[i].PlcUnitIndx = unitIU;
	var[i].unitType = unitPerc;
	var[i].DefaultUnit = UNIT_PERCENT;
	var[i].precision = 0;
	cfg->Param[i].min = 0.0;
	cfg->Param[i].max = 1.0;
	cfg->Param[i].incrMin = 0.01;
	cfg->Param[i].incrMax = 0.1;
	cfg->Param[i].defaultVal = 0.5;
	var[i].segm = 0;

	//////////////////////////////
	//	TIG Power Supply

	i = parTIG_AmpSP;
	strcpy(var[i].name , "PRIMARY ARC AMPS");
	strcpy(var[i].enumTXT, "parTIG_AmpSP");
	var[i].PlcUnitIndx = unitIU;
	var[i].unitType = unitAmp;
	var[i].DefaultUnit = UNIT_Amp;
	var[i].precision = 0;
	cfg->Param[i].min = 0.0;
	cfg->Param[i].max = 500.0;
	cfg->Param[i].incrMin = 1.0;
	cfg->Param[i].incrMax = 10.0;
	cfg->Param[i].defaultVal = 140.0;
	var[i].segm = 1;

	i = parTIG_AmpInSP;
	strcpy(var[i].name , "PRIMARY In ARC AMPS");
	strcpy(var[i].enumTXT, "parTIG_AmpInSP");
	var[i].PlcUnitIndx = unitIU;
	var[i].unitType = unitAmp;
	var[i].DefaultUnit = UNIT_Amp;
	var[i].precision = 0;
	cfg->Param[i].min = 0.0;
	cfg->Param[i].max = 500.0;
	cfg->Param[i].incrMin = 1.0;
	cfg->Param[i].incrMax = 10.0;
	cfg->Param[i].defaultVal = 140.0;
	var[i].segm = 1;

	i = parTIG_AmpOutSP;
	strcpy(var[i].name , "PRIMARY Out ARC AMPS");
	strcpy(var[i].enumTXT, "parTIG_AmpOutSP");
	var[i].PlcUnitIndx = unitIU;
	var[i].unitType = unitAmp;
	var[i].DefaultUnit = UNIT_Amp;
	var[i].precision = 0;
	cfg->Param[i].min = 0.0;
	cfg->Param[i].max = 500.0;
	cfg->Param[i].incrMin = 1.0;
	cfg->Param[i].incrMax = 10.0;
	cfg->Param[i].defaultVal = 140.0;
	var[i].segm = 1;

	i = parTIG_BackAmp;
	strcpy(var[i].name , "BACKGND ARC AMPS");
	strcpy(var[i].enumTXT, "parTIG_BackAmp");
	var[i].PlcUnitIndx = unitIU;
	var[i].unitType = unitAmp;
	var[i].DefaultUnit = UNIT_Amp;
	var[i].precision = 0;
	cfg->Param[i].min = 0.0;
	cfg->Param[i].max = 500.0;
	cfg->Param[i].incrMin = 1.0;
	cfg->Param[i].incrMax = 10.0;
	cfg->Param[i].defaultVal = 110.0;
	var[i].segm = 1;

	i = parTIG_Boost1;
	strcpy(var[i].name , "Boost1 ARC AMPS");
	strcpy(var[i].enumTXT, "parTIG_Boost1");
	var[i].PlcUnitIndx = unitIU;
	var[i].unitType = unitAmp;
	var[i].DefaultUnit = UNIT_Amp;
	var[i].precision = 0;
	cfg->Param[i].max = 500.0;
	cfg->Param[i].min = -cfg->Param[i].max;
	cfg->Param[i].incrMin = 1.0;
	cfg->Param[i].incrMax = 10.0;
	cfg->Param[i].defaultVal = 0.0;
	var[i].segm = 1;

	i = parTIG_Boost2;
	strcpy(var[i].name , "Boost2 ARC AMPS");
	strcpy(var[i].enumTXT, "parTIG_Boost2");
	var[i].PlcUnitIndx = unitIU;
	var[i].unitType = unitAmp;
	var[i].DefaultUnit = UNIT_Amp;
	var[i].precision = 0;
	cfg->Param[i].max = 500.0;
	cfg->Param[i].min = -cfg->Param[i].max;
	cfg->Param[i].incrMin = 1.0;
	cfg->Param[i].incrMax = 10.0;
	cfg->Param[i].defaultVal = 0.0;
	var[i].segm = 1;

	i = parTIG_PulseFreq;
	strcpy(var[i].name , "ARC AMPS FREQ.");
	strcpy(var[i].enumTXT, "parTIG_PulseFreq");
	var[i].PlcUnitIndx = unitIU;
	var[i].unitType = unitFreq;
	var[i].DefaultUnit = UNIT_Hz;
	var[i].precision = 1;
	cfg->Param[i].min = 0.0;
	cfg->Param[i].max = 100.0;
	cfg->Param[i].incrMin = 0.1;
	cfg->Param[i].incrMax = 1.0;
	cfg->Param[i].defaultVal = 10.0;
	var[i].segm = 1;

	i = parTIG_PulseWidth;
	strcpy(var[i].name , "ARC PULSE DUTY");
	strcpy(var[i].enumTXT, "parTIG_PulseWidth");
	var[i].PlcUnitIndx = unitIU;
	var[i].unitType = unitPerc;
	var[i].DefaultUnit = UNIT_PERCENT;
	var[i].precision = 0;
	cfg->Param[i].min = 0.001;
	cfg->Param[i].max = 1.0;
	cfg->Param[i].incrMin = 0.001;
	cfg->Param[i].incrMax = 0.1;
	cfg->Param[i].defaultVal = 0.5;
	var[i].segm = 1;

	i = parTIG_StartAmp;
	strcpy(var[i].name , "INITIAL ARC AMPS");
	strcpy(var[i].enumTXT, "parTIG_StartAmp");
	var[i].PlcUnitIndx = unitIU;
	var[i].unitType = unitAmp;
	var[i].DefaultUnit = UNIT_Amp;
	var[i].precision = 0;
	cfg->Param[i].min = 0.0;
	cfg->Param[i].max = 500.0;
	cfg->Param[i].incrMin = 1.0;
	cfg->Param[i].incrMax = 10.0;
	cfg->Param[i].defaultVal = 45.0;
	var[i].segm = 0;

	i = parTIG_EndAmp;
	strcpy(var[i].name , "FINAL ARC AMPS");
	strcpy(var[i].enumTXT, "parTIG_EndAmp");
	var[i].PlcUnitIndx = unitIU;
	var[i].unitType = unitAmp;
	var[i].DefaultUnit = UNIT_Amp;
	var[i].precision = 0;
	cfg->Param[i].min = 0.0;
	cfg->Param[i].max = 500.0;
	cfg->Param[i].incrMin = 1.0;
	cfg->Param[i].incrMax = 10.0;
	cfg->Param[i].defaultVal = 50.0;
	var[i].segm = 0;

	i = parTIG_RampUp;
	strcpy(var[i].name , "ARC AMP UPSLOPE TM");
	strcpy(var[i].enumTXT, "parTIG_RampUp");
	var[i].PlcUnitIndx = unitIU;
	var[i].unitType = unitTime;
	var[i].DefaultUnit = UNIT_sec;
	var[i].precision = 1;
	cfg->Param[i].min = 0.0;
	cfg->Param[i].max = 60.0;
	cfg->Param[i].incrMin = 0.1;
	cfg->Param[i].incrMax = 1.0;
	cfg->Param[i].defaultVal = 3.0;
	var[i].segm = 0;

	i = parTIG_RampDwn;
	strcpy(var[i].name , "AMPS DOWNSLOPE TM");
	strcpy(var[i].enumTXT, "parTIG_RampDwn");
	var[i].PlcUnitIndx = unitIU;
	var[i].unitType = unitTime;
	var[i].DefaultUnit = UNIT_sec;
	var[i].precision = 1;
	cfg->Param[i].min = 0.0;
	cfg->Param[i].max = 60.0;
	cfg->Param[i].incrMin = 0.1;
	cfg->Param[i].incrMax = 1.0;
	cfg->Param[i].defaultVal = 9.0;
	var[i].segm = 0;

	i = parTIG_StartDly;
	strcpy(var[i].name , "ARC AMP START DLY");
	strcpy(var[i].enumTXT, "parTIG_StartDly");
	var[i].PlcUnitIndx = unitIU;
	var[i].unitType = unitTime;
	var[i].DefaultUnit = UNIT_sec;
	var[i].precision = 1;
	cfg->Param[i].min = 0.0;
	cfg->Param[i].max = 10.0;
	cfg->Param[i].incrMin = 0.1;
	cfg->Param[i].incrMax = 1.0;
	cfg->Param[i].defaultVal = 2.0;
	var[i].segm = 0;

	i = parTIG_StopDly;
	strcpy(var[i].name , "AMPS DOWNSLOPE DLY");
	strcpy(var[i].enumTXT, "parTIG_StopDly");
	var[i].PlcUnitIndx = unitIU;
	var[i].unitType = unitTime;
	var[i].DefaultUnit = UNIT_sec;
	var[i].precision = 1;
	cfg->Param[i].min = 0.0;
	cfg->Param[i].max = 60.0;
	cfg->Param[i].incrMin = 0.1;
	cfg->Param[i].incrMax = 1.0;
	cfg->Param[i].defaultVal = 0.0;
	var[i].segm = 0;

	i = parTIG_CalibAmp1;
	strcpy(var[i].name , "TIG Calib Amp 1");
	strcpy(var[i].enumTXT, "parTIG_CalibAmp1");
	var[i].PlcUnitIndx = unitIU;
	var[i].unitType = unitAmp;
	var[i].DefaultUnit = UNIT_Amp;
	var[i].precision = 0;
	cfg->Param[i].min = 5.0;
	cfg->Param[i].max = 500.0;
	cfg->Param[i].incrMin = 1.0;
	cfg->Param[i].incrMax = 10.0;
	cfg->Param[i].defaultVal = 50.0;
	var[i].segm = 0;

	i = parTIG_CalibAmp2;
	strcpy(var[i].name , "TIG Calib Amp 2");
	strcpy(var[i].enumTXT, "parTIG_CalibAmp2");
	var[i].PlcUnitIndx = unitIU;
	var[i].unitType = unitAmp;
	var[i].DefaultUnit = UNIT_Amp;
	var[i].precision = 0;
	cfg->Param[i].min = 5.0;
	cfg->Param[i].max = 500.0;
	cfg->Param[i].incrMin = 1.0;
	cfg->Param[i].incrMax = 10.0;
	cfg->Param[i].defaultVal = 100.0;
	var[i].segm = 0;

	i = parTIG_AmpSP_Boost;
	strcpy(var[i].name , "TIG Amp Boost");
	strcpy(var[i].enumTXT, "parTIG_AmpSP_Boost");
	var[i].PlcUnitIndx = unitIU;
	var[i].unitType = unitPerc;
	var[i].DefaultUnit = UNIT_PERCENT;
	var[i].precision = 2;
	cfg->Param[i].min = -0.5;
	cfg->Param[i].max = 0.5;
	cfg->Param[i].incrMin = 0.05;
	cfg->Param[i].incrMax = 0.1;
	cfg->Param[i].defaultVal = 0.0;
	var[i].segm = 0;

	//////////////////////////////
	//	HW Power Supply

	i = parHW_AmpSP;
	strcpy(var[i].name , "HW PRIMARY AMPS");
	strcpy(var[i].enumTXT, "parHW_AmpSP");
	var[i].PlcUnitIndx = unitIU;
	var[i].unitType = unitAmp;
	var[i].DefaultUnit = UNIT_Amp;
	var[i].precision = 0;
	cfg->Param[i].min = 5.0;
	cfg->Param[i].max = 100.0;
	cfg->Param[i].incrMin = 1.0;
	cfg->Param[i].incrMax = 10.0;
	cfg->Param[i].defaultVal = 80.0;
	var[i].segm = 1;

	i = parHW_VoltSP;
	strcpy(var[i].name , "HW Volt SP");
	strcpy(var[i].enumTXT, "parHW_VoltSP");
	var[i].PlcUnitIndx = unitIU;
	var[i].unitType = unitVolt;
	var[i].DefaultUnit = UNIT_Volt;
	var[i].precision = 0;
	cfg->Param[i].min = 0.0;
	cfg->Param[i].max = 100.0;
	cfg->Param[i].incrMin = 1.0;
	cfg->Param[i].incrMax = 10.0;
	cfg->Param[i].defaultVal = 50.0;
	var[i].segm = 0;

	i = parHW_StartAmp;
	strcpy(var[i].name , "HW INITIAL AMPS");
	strcpy(var[i].enumTXT, "parHW_StartAmp");
	var[i].PlcUnitIndx = unitIU;
	var[i].unitType = unitAmp;
	var[i].DefaultUnit = UNIT_Amp;
	var[i].precision = 0;
	cfg->Param[i].min = 5.0;
	cfg->Param[i].max = 100.0;
	cfg->Param[i].incrMin = 1.0;
	cfg->Param[i].incrMax = 10.0;
	cfg->Param[i].defaultVal = 50.0;
	var[i].segm = 0;

	i = parHW_EndAmp;
	strcpy(var[i].name , "HW FINAL AMPS");
	strcpy(var[i].enumTXT, "parHW_EndAmp");
	var[i].PlcUnitIndx = unitIU;
	var[i].unitType = unitAmp;
	var[i].DefaultUnit = UNIT_Amp;
	var[i].precision = 0;
	cfg->Param[i].min = 5.0;
	cfg->Param[i].max = 100.0;
	cfg->Param[i].incrMin = 1.0;
	cfg->Param[i].incrMax = 10.0;
	cfg->Param[i].defaultVal = 50.0;
	var[i].segm = 0;

	i = parHW_RampUp;
	strcpy(var[i].name , "HW UPSLOPE TM");
	strcpy(var[i].enumTXT, "parHW_RampUp");
	var[i].PlcUnitIndx = unitIU;
	var[i].unitType = unitTime;
	var[i].DefaultUnit = UNIT_sec;
	var[i].precision = 1;
	cfg->Param[i].min = 0.0;
	cfg->Param[i].max = 60.0;
	cfg->Param[i].incrMin = 0.1;
	cfg->Param[i].incrMax = 1.0;
	cfg->Param[i].defaultVal = 3.0;
	var[i].segm = 0;

	i = parHW_RampDwn;
	strcpy(var[i].name , "HW DOWNSLOPE TM");
	strcpy(var[i].enumTXT, "parHW_RampDwn");
	var[i].PlcUnitIndx = unitIU;
	var[i].unitType = unitTime;
	var[i].DefaultUnit = UNIT_sec;
	var[i].precision = 1;
	cfg->Param[i].min = 0.0;
	cfg->Param[i].max = 60.0;
	cfg->Param[i].incrMin = 0.1;
	cfg->Param[i].incrMax = 1.0;
	cfg->Param[i].defaultVal = 0.5;
	var[i].segm = 0;

	i = parHW_RampUpDly;
	strcpy(var[i].name , "HW UPSLOPE DLY ");
	strcpy(var[i].enumTXT, "parHW_RampUpDly");
	var[i].PlcUnitIndx = unitIU;
	var[i].unitType = unitTime;
	var[i].DefaultUnit = UNIT_sec;
	var[i].precision = 1;
	cfg->Param[i].min = 0.0;
	cfg->Param[i].max = 60.0;
	cfg->Param[i].incrMin = 0.1;
	cfg->Param[i].incrMax = 1.0;
	cfg->Param[i].defaultVal = 8.0;
	var[i].segm = 0;

	i = parHW_RampDwnDly;
	strcpy(var[i].name , "HW DOWNSLOPE DLY");
	strcpy(var[i].enumTXT, "parHW_RampDwnDly");
	var[i].PlcUnitIndx = unitIU;
	var[i].unitType = unitTime;
	var[i].DefaultUnit = UNIT_sec;
	var[i].precision = 1;
	cfg->Param[i].min = 0.0;
	cfg->Param[i].max = 60.0;
	cfg->Param[i].incrMin = 0.1;
	cfg->Param[i].incrMax = 1.0;
	cfg->Param[i].defaultVal = 2.0;
	var[i].segm = 0;

	i = parHW_CalibAmp1;
	strcpy(var[i].name , "HW Calib Amp 1");
	strcpy(var[i].enumTXT, "parHW_CalibAmp1");
	var[i].PlcUnitIndx = unitIU;
	var[i].unitType = unitAmp;
	var[i].DefaultUnit = UNIT_Amp;
	var[i].precision = 0;
	cfg->Param[i].min = 5.0;
	cfg->Param[i].max = 160.0;
	cfg->Param[i].incrMin = 1.0;
	cfg->Param[i].incrMax = 10.0;
	cfg->Param[i].defaultVal = 25.0;
	var[i].segm = 0;

	i = parHW_CalibAmp2;
	strcpy(var[i].name , "HW Calib Amp 2");
	strcpy(var[i].enumTXT, "parHW_CalibAmp2");
	var[i].PlcUnitIndx = unitIU;
	var[i].unitType = unitAmp;
	var[i].DefaultUnit = UNIT_Amp;
	var[i].precision = 0;
	cfg->Param[i].min = 5.0;
	cfg->Param[i].max = 160.0;
	cfg->Param[i].incrMin = 1.0;
	cfg->Param[i].incrMax = 10.0;
	cfg->Param[i].defaultVal = 50.0;
	var[i].segm = 0;

	i = parHW_AmpSP_Boost;
	strcpy(var[i].name , "HW Amp Boost");
	strcpy(var[i].enumTXT, "parHW_AmpSP_Boost");
	var[i].PlcUnitIndx = unitIU;
	var[i].unitType = unitPerc;
	var[i].DefaultUnit = UNIT_PERCENT;
	var[i].precision = 2;
	cfg->Param[i].min = -0.5;
	cfg->Param[i].max = 0.5;
	cfg->Param[i].incrMin = 0.05;
	cfg->Param[i].incrMax = 0.1;
	cfg->Param[i].defaultVal = 0.0;
	var[i].segm = 0;

	/////////////////////////////
	// TVL

	i = parTVL_VelSP;
	strcpy(var[i].name , "TVL PRIMARY SPEED");
	strcpy(var[i].enumTXT, "parTVL_VelSP");
	var[i].PlcUnitIndx = unitIU;
	var[i].unitType = unitSpeed;
	var[i].DefaultUnit = UNIT_inch_per_min;
	var[i].precision = 0;
	cfg->Param[i].min = 0.0 *  in_min_2_mm_s;
	cfg->Param[i].max = 100.0 *  in_min_2_mm_s;
	cfg->Param[i].incrMin = 0.1 * in_min_2_mm_s;
	cfg->Param[i].incrMax = 10.0 * cfg->Param[i].incrMin;
	cfg->Param[i].defaultVal = 3.5 * in_min_2_mm_s;
	var[i].segm = 1;

	i = parTVL_VelInSP;
	strcpy(var[i].name , "TVL IN PRIMARY SPEED");
	strcpy(var[i].enumTXT, "parTVL_VelInSP");
	var[i].PlcUnitIndx = unitIU;
	var[i].unitType = unitSpeed;
	var[i].DefaultUnit = UNIT_inch_per_min;
	var[i].precision = 0;
	cfg->Param[i].min = 0.0 *  in_min_2_mm_s;
	cfg->Param[i].max = 100.0 *  in_min_2_mm_s;
	cfg->Param[i].incrMin = 0.1 * in_min_2_mm_s;
	cfg->Param[i].incrMax = 10.0 * cfg->Param[i].incrMin;
	cfg->Param[i].defaultVal = 3.5 * in_min_2_mm_s;
	var[i].segm = 1;

	i = parTVL_VelOutSP;
	strcpy(var[i].name , "TVL Out PRIMARY SPEED");
	strcpy(var[i].enumTXT, "parTVL_VelOutSP");
	var[i].PlcUnitIndx = unitIU;
	var[i].unitType = unitSpeed;
	var[i].DefaultUnit = UNIT_inch_per_min;
	var[i].precision = 0;
	cfg->Param[i].min = 0.0 *  in_min_2_mm_s;
	cfg->Param[i].max = 100.0 *  in_min_2_mm_s;
	cfg->Param[i].incrMin = 0.1 * in_min_2_mm_s;
	cfg->Param[i].incrMax = 10.0 * cfg->Param[i].incrMin;
	cfg->Param[i].defaultVal = 3.5 * in_min_2_mm_s;
	var[i].segm = 1;

	i = parTVL_VelBackSP;
	strcpy(var[i].name , "TVL Bckg SPEED");
	strcpy(var[i].enumTXT, "parTVL_VelBackSP");
	var[i].PlcUnitIndx = unitIU;
	var[i].unitType = unitSpeed;
	var[i].DefaultUnit = UNIT_inch_per_min;
	var[i].precision = 0;
	cfg->Param[i].min = 0.0 *  in_min_2_mm_s;
	cfg->Param[i].max = 100.0 *  in_min_2_mm_s;
	cfg->Param[i].incrMin = 0.1 * in_min_2_mm_s;
	cfg->Param[i].incrMax = 10.0 * cfg->Param[i].incrMin;
	cfg->Param[i].defaultVal = 3.5 * in_min_2_mm_s;
	var[i].segm = 1;

	i = parTVL_Boost1;
	strcpy(var[i].name , "TVL Boost1 SPEED");
	strcpy(var[i].enumTXT, "parTVL_Boost1");
	var[i].PlcUnitIndx = unitIU;
	var[i].unitType = unitSpeed;
	var[i].DefaultUnit = UNIT_inch_per_min;
	var[i].precision = 0;
	cfg->Param[i].max = 100.0 *  in_min_2_mm_s;
	cfg->Param[i].min = -cfg->Param[i].max;
	cfg->Param[i].incrMin = 0.1 * in_min_2_mm_s;
	cfg->Param[i].incrMax = 10.0 * cfg->Param[i].incrMin;
	cfg->Param[i].defaultVal = 0.0;
	var[i].segm = 1;

	i = parTVL_Boost2;
	strcpy(var[i].name , "TVL Boost2 SPEED");
	strcpy(var[i].enumTXT, "parTVL_Boost2");
	var[i].PlcUnitIndx = unitIU;
	var[i].unitType = unitSpeed;
	var[i].DefaultUnit = UNIT_inch_per_min;
	var[i].precision = 0;
	cfg->Param[i].max = 100.0 *  in_min_2_mm_s;
	cfg->Param[i].min = -cfg->Param[i].max;
	cfg->Param[i].incrMin = 0.1 * in_min_2_mm_s;
	cfg->Param[i].incrMax = 10.0 * cfg->Param[i].incrMin;
	cfg->Param[i].defaultVal = 0.0;
	var[i].segm = 1;

	i = parTVL_InitVel;
	strcpy(var[i].name , "TVL INITIAL SPEED");
	strcpy(var[i].enumTXT, "parTVL_InitVel");
	var[i].PlcUnitIndx = unitIU;
	var[i].unitType = unitSpeed;
	var[i].DefaultUnit = UNIT_inch_per_min;
	var[i].precision = 0;
	cfg->Param[i].min = 0.0;
	cfg->Param[i].max =  50.0* in_min_2_mm_s;
	cfg->Param[i].incrMin = 0.1 * in_min_2_mm_s;
	cfg->Param[i].incrMax = 10 * cfg->Param[i].incrMin;
	cfg->Param[i].defaultVal = 0.0 * in_min_2_mm_s;
	var[i].segm = 0;

	i = parTVL_FinalVel;
	strcpy(var[i].name , "TVL FINAL SPEED");
	strcpy(var[i].enumTXT, "parTVL_FinalVel");
	var[i].PlcUnitIndx = unitIU;
	var[i].unitType = unitSpeed;
	var[i].DefaultUnit = UNIT_inch_per_min;
	var[i].precision = 0;
	cfg->Param[i].min = 0.0;
	cfg->Param[i].max =  50.0 * in_min_2_mm_s;
	cfg->Param[i].incrMin = 0.1 * in_min_2_mm_s;
	cfg->Param[i].incrMax = 10 * cfg->Param[i].incrMin;
	cfg->Param[i].defaultVal = 1.0 * in_min_2_mm_s;
	var[i].segm = 0;

	i = parTVL_StartDly;
	strcpy(var[i].name , "TVL START DLY");
	strcpy(var[i].enumTXT, "parTVL_StartDly");
	var[i].PlcUnitIndx = unitIU;
	var[i].unitType = unitTime;
	var[i].DefaultUnit = UNIT_sec;
	var[i].precision = 1;
	cfg->Param[i].min = 0.0;
	cfg->Param[i].max = 60.0;
	cfg->Param[i].incrMin = 0.1;
	cfg->Param[i].incrMax = 1.0;
	cfg->Param[i].defaultVal = 5.0;
	var[i].segm = 0;

	i = parTVL_RampUp;
	strcpy(var[i].name , "TVL UPSLOPE TM");
	strcpy(var[i].enumTXT, "parTVL_RampUp");
	var[i].PlcUnitIndx = unitIU;
	var[i].unitType = unitTime;
	var[i].DefaultUnit = UNIT_sec;
	var[i].precision = 1;
	cfg->Param[i].min = 0.0;
	cfg->Param[i].max = 60.0;
	cfg->Param[i].incrMin = 0.1;
	cfg->Param[i].incrMax = 1.0;
	cfg->Param[i].defaultVal = 0.0;
	var[i].segm = 0;

	i = parTVL_StopDly;
	strcpy(var[i].name , "TVL DOWNSLOPE DLY");
	strcpy(var[i].enumTXT, "parTVL_StopDly");
	var[i].PlcUnitIndx = unitIU;
	var[i].unitType = unitTime;
	var[i].DefaultUnit = UNIT_sec;
	var[i].precision = 1;
	cfg->Param[i].min = 0.0;
	cfg->Param[i].max = 60.0;
	cfg->Param[i].incrMin = 0.1;
	cfg->Param[i].incrMax = 1.0;
	cfg->Param[i].defaultVal = 10.0;
	var[i].segm = 0;

	i = parTVL_RampDwn;
	strcpy(var[i].name , "TVL DOWNSLOPE TM");
	strcpy(var[i].enumTXT, "parTVL_RampDwn");
	var[i].PlcUnitIndx = unitIU;
	var[i].unitType = unitTime;
	var[i].DefaultUnit = UNIT_sec;
	var[i].precision = 1;
	cfg->Param[i].min = 0.0;
	cfg->Param[i].max = 60.0;
	cfg->Param[i].incrMin = 0.1;
	cfg->Param[i].incrMax = 1.0;
	cfg->Param[i].defaultVal = 0.0;
	var[i].segm = 0;

	i = parTVL_RampUpdate;
	strcpy(var[i].name , "TVL Ramp Update");
	strcpy(var[i].enumTXT, "parTVL_RampUpdate");
	var[i].PlcUnitIndx = unitIU;
	var[i].unitType = unitTime;
	var[i].DefaultUnit = UNIT_sec;
	var[i].precision = 1;
	cfg->Param[i].min = 0.0;
	cfg->Param[i].max = 60.0;
	cfg->Param[i].incrMin = 0.1;
	cfg->Param[i].incrMax = 1.0;
	cfg->Param[i].defaultVal = 0.1;
	var[i].segm = 0;

	i = parTVL_JogSpeedDirCntrl;
	strcpy(var[i].name , "TVL Jog Speed");
	strcpy(var[i].enumTXT, "parTVL_JogSpeedDirCntrl");
	var[i].PlcUnitIndx = unitIU;
	var[i].unitType = unitPerc;
	var[i].DefaultUnit = UNIT_PERCENT;
	var[i].precision = 0;
	cfg->Param[i].min = 0.0;
	cfg->Param[i].max = 1.0;
	cfg->Param[i].incrMin = 0.01;
	cfg->Param[i].incrMax = 0.1;
	cfg->Param[i].defaultVal = 1.0;
	var[i].segm = 0;

	i = parTVL_RunDist;
	//strcpy(var[i].name , "RUN Segments");
	strcpy(var[i].name , "RUN Dist.");
	strcpy(var[i].enumTXT, "parTVL_RunDist");
	var[i].PlcUnitIndx = unitIU;
	var[i].unitType =  unitIU;
	var[i].DefaultUnit = unitIU;
	var[i].precision = 0;
	cfg->Param[i].min = 0.0;
	cfg->Param[i].max = 100000.0;
	cfg->Param[i].incrMin = 1;
	cfg->Param[i].incrMax = 1000;
	cfg->Param[i].defaultVal = 40;
	var[i].segm = 0;

	i = parTVL_ZigZagDist;
	//strcpy(var[i].name , "RUN Segments");
	strcpy(var[i].name , "Zig Zag Dist.");
	strcpy(var[i].enumTXT, "parTVL_ZigZagDist");
	var[i].PlcUnitIndx = unitIU;
	var[i].unitType =  unitIU;
	var[i].DefaultUnit = unitIU;
	var[i].precision = 0;
	cfg->Param[i].min = 0.0;
	cfg->Param[i].max = 1000.0;
	cfg->Param[i].incrMin = 1;
	cfg->Param[i].incrMax = 10;
	cfg->Param[i].defaultVal = 0;
	var[i].segm = 0;

	i = parTVL_BalanceDist;
	strcpy(var[i].name , "A/B Balance Dist.");
	strcpy(var[i].enumTXT, "parTVL_BalanceDist");
	var[i].PlcUnitIndx = unitIU;
	var[i].unitType =  unitIU;
	var[i].DefaultUnit = unitIU;
	var[i].precision = 0;
	cfg->Param[i].min = -1000.0;
	cfg->Param[i].max = 1000.0;
	cfg->Param[i].incrMin = 1;
	cfg->Param[i].incrMax = 10;
	cfg->Param[i].defaultVal = 0;
	var[i].segm = 0;

	i = parTVL_RewrapDly;
	strcpy(var[i].name , "TVL REWRAP DLY");
	strcpy(var[i].enumTXT, "parTVL_RewrapDly");
	var[i].PlcUnitIndx = unitIU;
	var[i].unitType = unitTime;
	var[i].DefaultUnit = UNIT_sec;
	var[i].precision = 1;
	cfg->Param[i].min = 0.0;
	cfg->Param[i].max = 300.0;
	cfg->Param[i].incrMin = 0.1;
	cfg->Param[i].incrMax = 1.0;
	cfg->Param[i].defaultVal = 2.0;
	var[i].segm = 0;

	i = parTVL_OverlapDist;
	strcpy(var[i].name , "TVL Overlap ");
	strcpy(var[i].enumTXT, "parTVL_OverlapDist");
	var[i].PlcUnitIndx = unitIU;
	var[i].unitType =  unitIU;
	var[i].DefaultUnit = unitIU;
	var[i].precision = 0;
	cfg->Param[i].min = -300000.0;
	cfg->Param[i].max = 300000.0;
	cfg->Param[i].incrMin = 1;
	cfg->Param[i].incrMax = 1;
	cfg->Param[i].defaultVal = 0;
	var[i].segm = 0;

	i = parTVL_RewrapVel;
	strcpy(var[i].name , "TVL REWRAP SP");
	strcpy(var[i].enumTXT, "parTVL_RewrapVel");
	var[i].PlcUnitIndx = unitIU;
	var[i].unitType = unitSpeed;
	var[i].DefaultUnit = UNIT_inch_per_min;
	var[i].precision = 0;
	cfg->Param[i].min = 0.0;
	cfg->Param[i].max = 110.0 * in_min_2_mm_s;
	cfg->Param[i].incrMin = 0.1 * in_min_2_mm_s;
	cfg->Param[i].incrMax = 10.0 * cfg->Param[i].incrMin;
	cfg->Param[i].defaultVal = 10.0;
	var[i].segm = 0;

	i = parTVL_Jog2Stop;
	strcpy(var[i].name , "TVL Jog2Stop");
	strcpy(var[i].enumTXT, "parTVL_Jog2Stop");
	var[i].PlcUnitIndx = unitIU;
	var[i].unitType = unitSpeed;
	var[i].DefaultUnit = UNIT_inch_per_min;
	var[i].precision = 2;
	cfg->Param[i].min = 0.0;
	cfg->Param[i].max = 4.5;
	cfg->Param[i].incrMin = 0.1 * in_min_2_mm_s;
	cfg->Param[i].incrMax = 1.0;
	cfg->Param[i].defaultVal = 1.5;
	var[i].segm = 0;

	i = parTVL_CalibVel1;
	strcpy(var[i].name , "TVL Calib Speed 1");
	strcpy(var[i].enumTXT, "parTVL_CalibVel1");
	var[i].PlcUnitIndx = unitIU;
	var[i].unitType = unitSpeed;
	var[i].DefaultUnit = UNIT_inch_per_min;
	var[i].precision = 0;
	cfg->Param[i].min = 1.0 *  in_min_2_mm_s;
	cfg->Param[i].max = 100.0 *  in_min_2_mm_s;
	cfg->Param[i].incrMin = 0.1 * in_min_2_mm_s;
	cfg->Param[i].incrMax = 10.0 * cfg->Param[i].incrMin;
	cfg->Param[i].defaultVal = 3.0 * in_min_2_mm_s;
	var[i].segm = 0;

	i = parTVL_CalibVel2;
	strcpy(var[i].name , "TVL Calib Speed 2");
	strcpy(var[i].enumTXT, "parTVL_CalibVel2");
	var[i].PlcUnitIndx = unitIU;
	var[i].unitType = unitSpeed;
	var[i].DefaultUnit = UNIT_inch_per_min;
	var[i].precision = 0;
	cfg->Param[i].min = 1.0 *  in_min_2_mm_s;
	cfg->Param[i].max = 100.0 *  in_min_2_mm_s;
	cfg->Param[i].incrMin = 0.1 * in_min_2_mm_s;
	cfg->Param[i].incrMax = 10.0 * cfg->Param[i].incrMin;
	cfg->Param[i].defaultVal = 6.0 * in_min_2_mm_s;
	var[i].segm = 0;

	i = parTVL_TrackDia;
	strcpy(var[i].name , "Tungsten Track Dia");
	strcpy(var[i].enumTXT, "parTVL_TrackDia");
	var[i].PlcUnitIndx = unitIU;
	var[i].unitType = unitLength;
	var[i].DefaultUnit = UNIT_inch;
	var[i].precision = 1;
	cfg->Param[i].min = 1.0 * in_2_mm;
	cfg->Param[i].max = 200.0 * in_2_mm;
	cfg->Param[i].incrMin = 0.01 * in_2_mm;
	cfg->Param[i].incrMax = 1.0 * in_2_mm;
	cfg->Param[i].defaultVal = 4.5 * in_2_mm;
	var[i].segm = 0;

	i = parTVL_SpeedTolerane;
	strcpy(var[i].name , "TVL Speed Tolerance");
	strcpy(var[i].enumTXT, "parTVL_SpeedTolerane");
	var[i].PlcUnitIndx = unitIU;
	var[i].unitType = unitPerc;
	var[i].DefaultUnit = UNIT_PERCENT;
	var[i].precision = 0;
	cfg->Param[i].min = 0.0;
	cfg->Param[i].max = 5.0;
	cfg->Param[i].incrMin = 0.01;
	cfg->Param[i].incrMax = 0.1;
	cfg->Param[i].defaultVal = 5.0;
	var[i].segm = 0;

	///////////////////////////////

	i = parCONTIN_TVL_RampDwn;
	strcpy(var[i].name , "CONTIN_TVL_RampDwn");
	strcpy(var[i].enumTXT, "parCONTIN_TVL_RampDwn");
	var[i].PlcUnitIndx = unitIU;
	var[i].unitType = unitTime;
	var[i].DefaultUnit = UNIT_sec;
	var[i].precision = 1;
	cfg->Param[i].min = 0.0;
	cfg->Param[i].max = 60.0;
	cfg->Param[i].incrMin = 0.1;
	cfg->Param[i].incrMax = 1.0;
	cfg->Param[i].defaultVal = 0.0;
	var[i].segm = 0;

	i = parCONTIN_TVL_RampUp;
	strcpy(var[i].name , "CONTIN_TVL_RampUp");
	strcpy(var[i].enumTXT, "parCONTIN_TVL_RampUp");
	var[i].PlcUnitIndx = unitIU;
	var[i].unitType = unitTime;
	var[i].DefaultUnit = UNIT_sec;
	var[i].precision = 1;
	cfg->Param[i].min = 0.0;
	cfg->Param[i].max = 60.0;
	cfg->Param[i].incrMin = 0.1;
	cfg->Param[i].incrMax = 1.0;
	cfg->Param[i].defaultVal = 0.0;
	var[i].segm = 0;

	i = parCONTIN_WF_RampDwn;
	strcpy(var[i].name , "CONTIN_WF_RampDwn");
	strcpy(var[i].enumTXT, "parCONTIN_WF_RampDwn");
	var[i].PlcUnitIndx = unitIU;
	var[i].unitType = unitTime;
	var[i].DefaultUnit = UNIT_sec;
	var[i].precision = 1;
	cfg->Param[i].min = 0.0;
	cfg->Param[i].max = 60.0;
	cfg->Param[i].incrMin = 0.1;
	cfg->Param[i].incrMax = 1.0;
	cfg->Param[i].defaultVal = 0.0;
	var[i].segm = 0;

	i = parCONTIN_WF_RampUp;
	strcpy(var[i].name , "CONTIN_WF_RampUp");
	strcpy(var[i].enumTXT, "parCONTIN_WF_RampUp");
	var[i].PlcUnitIndx = unitIU;
	var[i].unitType = unitTime;
	var[i].DefaultUnit = UNIT_sec;
	var[i].precision = 1;
	cfg->Param[i].min = 0.0;
	cfg->Param[i].max = 60.0;
	cfg->Param[i].incrMin = 0.1;
	cfg->Param[i].incrMax = 1.0;
	cfg->Param[i].defaultVal = 0.0;
	var[i].segm = 0;

	i = parCONTIN_WP_RampDwn;
	strcpy(var[i].name , "CONTIN_WP_RampDwn");
	strcpy(var[i].enumTXT, "parCONTIN_WP_RampDwn");
	var[i].PlcUnitIndx = unitIU;
	var[i].unitType = unitTime;
	var[i].DefaultUnit = UNIT_sec;
	var[i].precision = 1;
	cfg->Param[i].min = 0.0;
	cfg->Param[i].max = 60.0;
	cfg->Param[i].incrMin = 0.1;
	cfg->Param[i].incrMax = 1.0;
	cfg->Param[i].defaultVal = 0.0;
	var[i].segm = 0;

	i = parCONTIN_WP_RampUp;
	strcpy(var[i].name , "CONTIN_WP_RampUp");
	strcpy(var[i].enumTXT, "parCONTIN_WP_RampUp");
	var[i].PlcUnitIndx = unitIU;
	var[i].unitType = unitTime;
	var[i].DefaultUnit = UNIT_sec;
	var[i].precision = 1;
	cfg->Param[i].min = 0.0;
	cfg->Param[i].max = 60.0;
	cfg->Param[i].incrMin = 0.1;
	cfg->Param[i].incrMax = 1.0;
	cfg->Param[i].defaultVal = 0.0;
	var[i].segm = 0;

	i = parCONTIN_TIG_RampUp;
	strcpy(var[i].name , "parCONTIN_TIG_RampUp");
	strcpy(var[i].enumTXT, "parCONTIN_TIG_RampUp");
	var[i].PlcUnitIndx = unitIU;
	var[i].unitType = unitTime;
	var[i].DefaultUnit = UNIT_sec;
	var[i].precision = 1;
	cfg->Param[i].min = 0.0;
	cfg->Param[i].max = 60.0;
	cfg->Param[i].incrMin = 0.1;
	cfg->Param[i].incrMax = 1.0;
	cfg->Param[i].defaultVal = 0.0;
	var[i].segm = 0;

	i = parCONTIN_TIG_RampDwn;
	strcpy(var[i].name , "parCONTIN_TIG_RampDwn");
	strcpy(var[i].enumTXT, "parCONTIN_TIG_RampDwn");
	var[i].PlcUnitIndx = unitIU;
	var[i].unitType = unitTime;
	var[i].DefaultUnit = UNIT_sec;
	var[i].precision = 1;
	cfg->Param[i].min = 0.0;
	cfg->Param[i].max = 60.0;
	cfg->Param[i].incrMin = 0.1;
	cfg->Param[i].incrMax = 1.0;
	cfg->Param[i].defaultVal = 0.0;
	var[i].segm = 0;

	i = parCONTIN_TIG_Dwell;
	strcpy(var[i].name , "parCONTIN_TIG_Dwell");
	strcpy(var[i].enumTXT, "parCONTIN_TIG_Dwell");
	var[i].PlcUnitIndx = unitIU;
	var[i].unitType = unitTime;
	var[i].DefaultUnit = UNIT_sec;
	var[i].precision = 1;
	cfg->Param[i].min = 0.0;
	cfg->Param[i].max = 60.0;
	cfg->Param[i].incrMin = 0.1;
	cfg->Param[i].incrMax = 1.0;
	cfg->Param[i].defaultVal = 0.0;
	var[i].segm = 0;

	i = parCONTIN_TIG_Percent;
	strcpy(var[i].name , "parCONTIN_TIG_Percent");
	strcpy(var[i].enumTXT, "parCONTIN_TIG_Percent");
	var[i].PlcUnitIndx = unitIU;
	var[i].unitType = unitPerc;
	var[i].DefaultUnit = UNIT_PERCENT;
	var[i].precision = 0;
	cfg->Param[i].min = -0.8;
	cfg->Param[i].max = 0.8;
	cfg->Param[i].incrMin = 0.005;
	cfg->Param[i].incrMax = 0.01;
	cfg->Param[i].defaultVal = 0.0;
	var[i].segm = 0;

	/////////////////////////////
	// GAS

	i = parGAS_PrePurgeTm;
	strcpy(var[i].name , "GAS PREPURGE TM");
	strcpy(var[i].enumTXT, "parGAS_PrePurgeTm");
	var[i].PlcUnitIndx = unitIU;
	var[i].unitType = unitTime;
	var[i].DefaultUnit = UNIT_sec;
	var[i].precision = 1;
	cfg->Param[i].min = 0.0;
	cfg->Param[i].max = 60.0;
	cfg->Param[i].incrMin = 0.1;
	cfg->Param[i].incrMax = 1.0;
	cfg->Param[i].defaultVal = 2.0;
	var[i].segm = 0;

	i = parGAS_PostPurgeTm;
	strcpy(var[i].name , "GAS POSTPURGE TM");
	strcpy(var[i].enumTXT, "parGAS_PostPurgeTm");
	var[i].PlcUnitIndx = unitIU;
	var[i].unitType = unitTime;
	var[i].DefaultUnit = UNIT_sec;
	var[i].precision = 1;
	cfg->Param[i].min = 0.0;
	cfg->Param[i].max = 180.0;
	cfg->Param[i].incrMin = 0.1;
	cfg->Param[i].incrMax = 1.0;
	cfg->Param[i].defaultVal = 12.0;
	var[i].segm = 0;

	i = parGAS_Tmo;
	strcpy(var[i].name , "Gas On/Off TimeOut");
	strcpy(var[i].enumTXT, "parGAS_Tmo");
	var[i].PlcUnitIndx = unitIU;
	var[i].unitType = unitTime;
	var[i].DefaultUnit = UNIT_sec;
	var[i].precision = 1;
	cfg->Param[i].min = 0.0;
	cfg->Param[i].max = 5.0;
	cfg->Param[i].incrMin = 0.1;
	cfg->Param[i].incrMax = 1.0;
	cfg->Param[i].defaultVal = 3.0;
	var[i].segm = 0;

	/////////////////////////////
	// COOLANT
```
